PROGRAM P21_AL_WN
VAR
	//Analog Deviation Check
	Dev00, Dev01, Dev02, Dev03, Dev04, Dev05, Dev06, Dev07, Dev08, Dev09: FB_DeviationCheck;
	Dev10, Dev11, Dev12, Dev13, Dev14, Dev15, Dev16, Dev17, Dev18, Dev19: FB_DeviationCheck;
	Dev20, Dev21, Dev22, Dev23, Dev24, Dev25, Dev26, Dev27, Dev28, Dev29: FB_DeviationCheck;
		
	//Digital Noise Check
	wNoiseCheckTime: WORD := 100;	
	FB_AL32, FB_AL33, FB_AL34, FB_AL35, FB_AL36, FB_AL37, FB_AL38, FB_AL39: FB_NoiseCheck;	 
	FB_AL40, FB_AL41, FB_AL42, FB_AL43, FB_AL44, FB_AL45, FB_AL46, FB_AL47: FB_NoiseCheck;
	FB_AL48, FB_AL49, FB_AL50, FB_AL51, FB_AL52, FB_AL53, FB_AL54, FB_AL55: FB_NoiseCheck; 
	FB_AL56, FB_AL57, FB_AL58, FB_AL59, FB_AL60, FB_AL61, FB_AL62, FB_AL63: FB_NoiseCheck; 
	FB_AL64, FB_AL65, FB_AL66, FB_AL67, FB_AL68, FB_AL69, FB_AL70, FB_AL71: FB_NoiseCheck; 
	FB_AL72, FB_AL73, FB_AL74, FB_AL75, FB_AL76, FB_AL77, FB_AL78, FB_AL79: FB_NoiseCheck; 
	FB_AL80, FB_AL81, FB_AL82, FB_AL83, FB_AL84, FB_AL85, FB_AL86, FB_AL87: FB_NoiseCheck;
	FB_AL88, FB_AL89, FB_AL90, FB_AL91, FB_AL92, FB_AL93, FB_AL94, FB_AL95: FB_NoiseCheck; 
	FB_AL96, FB_AL97, FB_AL98, FB_AL99, FB_AL100, FB_AL101, FB_AL102, FB_AL103: FB_NoiseCheck; 
	FB_AL104, FB_AL105, FB_AL106, FB_AL107, FB_AL108, FB_AL109, FB_AL110, FB_AL111: FB_NoiseCheck;
	//FB_AL112, FB_AL113, FB_AL114, FB_AL115, FB_AL116, FB_AL117, FB_AL118, FB_AL119: FB_NoiseCheck; 
	FB_AL120, FB_AL121, FB_AL122, FB_AL123, FB_AL124, FB_AL125, FB_AL126, FB_AL127: FB_NoiseCheck;
	FB_AL128, FB_AL129, FB_AL130, FB_AL131, FB_AL132, FB_AL133, FB_AL134, FB_AL135: FB_NoiseCheck;
	FB_AL136, FB_AL137, FB_AL138, FB_AL139, FB_AL140, FB_AL141, FB_AL142, FB_AL143: FB_NoiseCheck;
	//FB_AL144, FB_AL145, FB_AL146, FB_AL147, FB_AL148, FB_AL149, FB_AL150, FB_AL151: FB_NoiseCheck;
	//FB_AL152, FB_AL153, FB_AL154, FB_AL155, FB_AL156, FB_AL157, FB_AL158, FB_AL159: FB_NoiseCheck;	
			
	FB_WN32, FB_WN33, FB_WN34, FB_WN35, FB_WN36, FB_WN37, FB_WN38, FB_WN39: FB_NoiseCheck; 
	FB_WN40, FB_WN41, FB_WN42, FB_WN43, FB_WN44, FB_WN45, FB_WN46, FB_WN47, FB_WN48, FB_WN49: FB_NoiseCheck; 
	FB_WN50, FB_WN51, FB_WN52, FB_WN53, FB_WN54, FB_WN55, FB_WN56, FB_WN57, FB_WN58, FB_WN59: FB_NoiseCheck; 
	FB_WN60, FB_WN61, FB_WN62, FB_WN63: FB_NoiseCheck;
									
	i: INT;
	bReset: BOOL;
	P_AL_Trig: R_TRIG;
	P_WN_Trig: R_TRIG;
	
	P_di_RST: R_TRIG;
		
	//Real Address
	n_AL_WORD AT%MB38: ARRAY[0..8] OF WORD; //16Bit
	n_WN_DWORD AT%MB56: ARRAY[0..1] OF DWORD; //32Bit
		
	n_AL_WORD_OLD: ARRAY[0..8] OF DWORD; //128EA
	n_WN_DWORD_OLD: ARRAY[0..1] OF DWORD; //64EA
	
	T1S_WN: TON;
	n_BZ_Order: ARRAY[0..1] OF BYTE;//부저 울림 순서, 1 -> Warning, 2 -> Alarm, 1 + 2 = 3 -> Alarm

END_VAR

A_AL_WN_Check();
D_AL_Check();
D_WN_Check();

is_AL := n_AL_WORD[0] > 0 OR n_AL_WORD[1] > 0 OR n_AL_WORD[2] > 0 OR n_AL_WORD[3] > 0 OR n_AL_WORD[4] > 0 OR
		 n_AL_WORD[5] > 0 OR n_AL_WORD[6] > 0 OR n_AL_WORD[7] > 0 OR n_AL_WORD[8] > 0;

is_WN := n_WN_DWORD[0] > 0 OR n_WN_DWORD[1] > 0 ;

//Alarm Processing
D_AL_Check();

//Alarm & Warning Reset
bReset := s_cm_RST;
 IF bReset THEN
	 s_is_DOR_Broken := 0;
 END_IF

//New AL Check
P_AL_Trig(CLK:= n_AL_WORD[0] > n_AL_WORD_OLD[0] OR n_AL_WORD[1] > n_AL_WORD_OLD[1] OR 
			  n_AL_WORD[2] > n_AL_WORD_OLD[2] OR n_AL_WORD[3] > n_AL_WORD_OLD[3] OR
			  n_AL_WORD[4] > n_AL_WORD_OLD[4] OR n_AL_WORD[5] > n_AL_WORD_OLD[5] OR
			  n_AL_WORD[6] > n_AL_WORD_OLD[6] OR n_AL_WORD[7] > n_AL_WORD_OLD[7] OR
			  n_AL_WORD[8] > n_AL_WORD_OLD[8]);
//New WN Check	
P_WN_Trig(CLK:= n_WN_DWORD[0] > n_WN_DWORD_OLD[0] OR n_WN_DWORD[1] > n_WN_DWORD_OLD[1]);

P_di_RST(CLK:= di_RST);	

//AL Backup	
FOR i := 0 TO 8 DO
	n_AL_WORD_OLD[i] := n_AL_WORD[i];
END_FOR
//WN Backup
FOR i := 0 TO 1 DO
	n_WN_DWORD_OLD[i] := n_WN_DWORD[i];
END_FOR

ACTION A_AL_WN_Check:
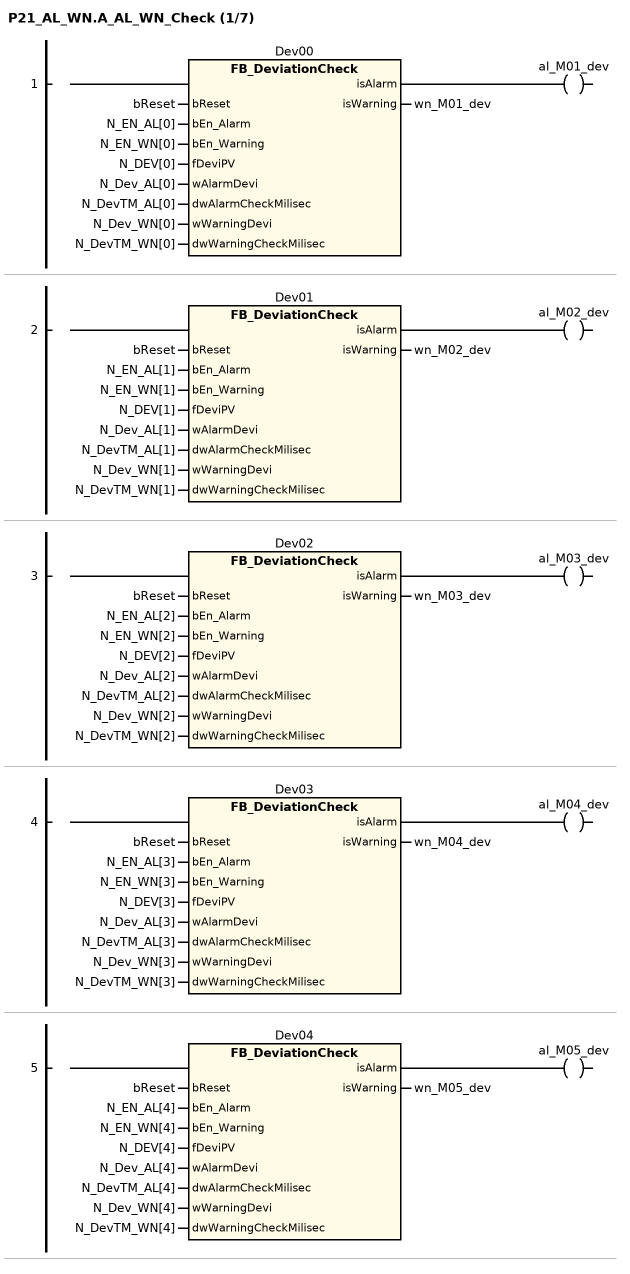
// NETWORK 1
Dev00(
    bReset := bReset,
    bEn_Alarm := N_EN_AL[0],
    bEn_Warning := N_EN_WN[0],
    fDeviPV := N_DEV[0],
    wAlarmDevi := N_Dev_AL[0],
    dwAlarmCheckMilisec := N_DevTM_AL[0],
    wWarningDevi := N_Dev_WN[0],
    dwWarningCheckMilisec := N_DevTM_WN[0],
    isWarning => wn_M01_dev); // FB_DeviationCheck
al_M01_dev := Dev00.isAlarm;

// NETWORK 2
Dev01(
    bReset := bReset,
    bEn_Alarm := N_EN_AL[1],
    bEn_Warning := N_EN_WN[1],
    fDeviPV := N_DEV[1],
    wAlarmDevi := N_Dev_AL[1],
    dwAlarmCheckMilisec := N_DevTM_AL[1],
    wWarningDevi := N_Dev_WN[1],
    dwWarningCheckMilisec := N_DevTM_WN[1],
    isWarning => wn_M02_dev); // FB_DeviationCheck
al_M02_dev := Dev01.isAlarm;

// NETWORK 3
Dev02(
    bReset := bReset,
    bEn_Alarm := N_EN_AL[2],
    bEn_Warning := N_EN_WN[2],
    fDeviPV := N_DEV[2],
    wAlarmDevi := N_Dev_AL[2],
    dwAlarmCheckMilisec := N_DevTM_AL[2],
    wWarningDevi := N_Dev_WN[2],
    dwWarningCheckMilisec := N_DevTM_WN[2],
    isWarning => wn_M03_dev); // FB_DeviationCheck
al_M03_dev := Dev02.isAlarm;

// NETWORK 4
Dev03(
    bReset := bReset,
    bEn_Alarm := N_EN_AL[3],
    bEn_Warning := N_EN_WN[3],
    fDeviPV := N_DEV[3],
    wAlarmDevi := N_Dev_AL[3],
    dwAlarmCheckMilisec := N_DevTM_AL[3],
    wWarningDevi := N_Dev_WN[3],
    dwWarningCheckMilisec := N_DevTM_WN[3],
    isWarning => wn_M04_dev); // FB_DeviationCheck
al_M04_dev := Dev03.isAlarm;

// NETWORK 5
Dev04(
    bReset := bReset,
    bEn_Alarm := N_EN_AL[4],
    bEn_Warning := N_EN_WN[4],
    fDeviPV := N_DEV[4],
    wAlarmDevi := N_Dev_AL[4],
    dwAlarmCheckMilisec := N_DevTM_AL[4],
    wWarningDevi := N_Dev_WN[4],
    dwWarningCheckMilisec := N_DevTM_WN[4],
    isWarning => wn_M05_dev); // FB_DeviationCheck
al_M05_dev := Dev04.isAlarm;

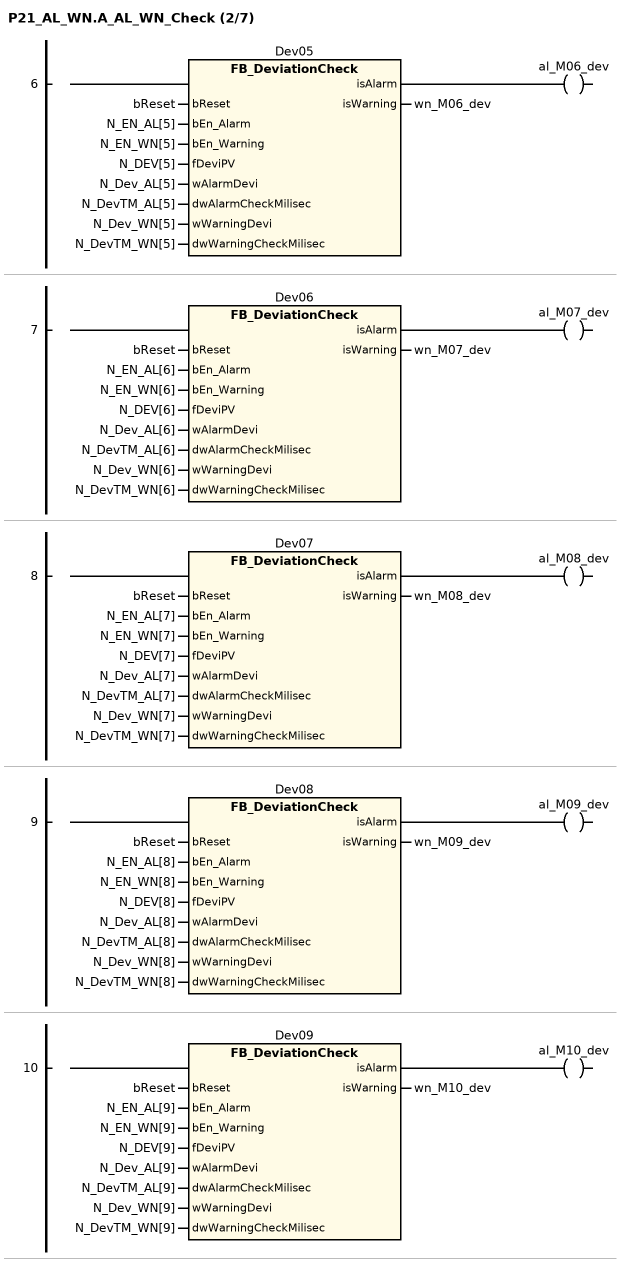
// NETWORK 6
Dev05(
    bReset := bReset,
    bEn_Alarm := N_EN_AL[5],
    bEn_Warning := N_EN_WN[5],
    fDeviPV := N_DEV[5],
    wAlarmDevi := N_Dev_AL[5],
    dwAlarmCheckMilisec := N_DevTM_AL[5],
    wWarningDevi := N_Dev_WN[5],
    dwWarningCheckMilisec := N_DevTM_WN[5],
    isWarning => wn_M06_dev); // FB_DeviationCheck
al_M06_dev := Dev05.isAlarm;

// NETWORK 7
Dev06(
    bReset := bReset,
    bEn_Alarm := N_EN_AL[6],
    bEn_Warning := N_EN_WN[6],
    fDeviPV := N_DEV[6],
    wAlarmDevi := N_Dev_AL[6],
    dwAlarmCheckMilisec := N_DevTM_AL[6],
    wWarningDevi := N_Dev_WN[6],
    dwWarningCheckMilisec := N_DevTM_WN[6],
    isWarning => wn_M07_dev); // FB_DeviationCheck
al_M07_dev := Dev06.isAlarm;

// NETWORK 8
Dev07(
    bReset := bReset,
    bEn_Alarm := N_EN_AL[7],
    bEn_Warning := N_EN_WN[7],
    fDeviPV := N_DEV[7],
    wAlarmDevi := N_Dev_AL[7],
    dwAlarmCheckMilisec := N_DevTM_AL[7],
    wWarningDevi := N_Dev_WN[7],
    dwWarningCheckMilisec := N_DevTM_WN[7],
    isWarning => wn_M08_dev); // FB_DeviationCheck
al_M08_dev := Dev07.isAlarm;

// NETWORK 9
Dev08(
    bReset := bReset,
    bEn_Alarm := N_EN_AL[8],
    bEn_Warning := N_EN_WN[8],
    fDeviPV := N_DEV[8],
    wAlarmDevi := N_Dev_AL[8],
    dwAlarmCheckMilisec := N_DevTM_AL[8],
    wWarningDevi := N_Dev_WN[8],
    dwWarningCheckMilisec := N_DevTM_WN[8],
    isWarning => wn_M09_dev); // FB_DeviationCheck
al_M09_dev := Dev08.isAlarm;

// NETWORK 10
Dev09(
    bReset := bReset,
    bEn_Alarm := N_EN_AL[9],
    bEn_Warning := N_EN_WN[9],
    fDeviPV := N_DEV[9],
    wAlarmDevi := N_Dev_AL[9],
    dwAlarmCheckMilisec := N_DevTM_AL[9],
    wWarningDevi := N_Dev_WN[9],
    dwWarningCheckMilisec := N_DevTM_WN[9],
    isWarning => wn_M10_dev); // FB_DeviationCheck
al_M10_dev := Dev09.isAlarm;

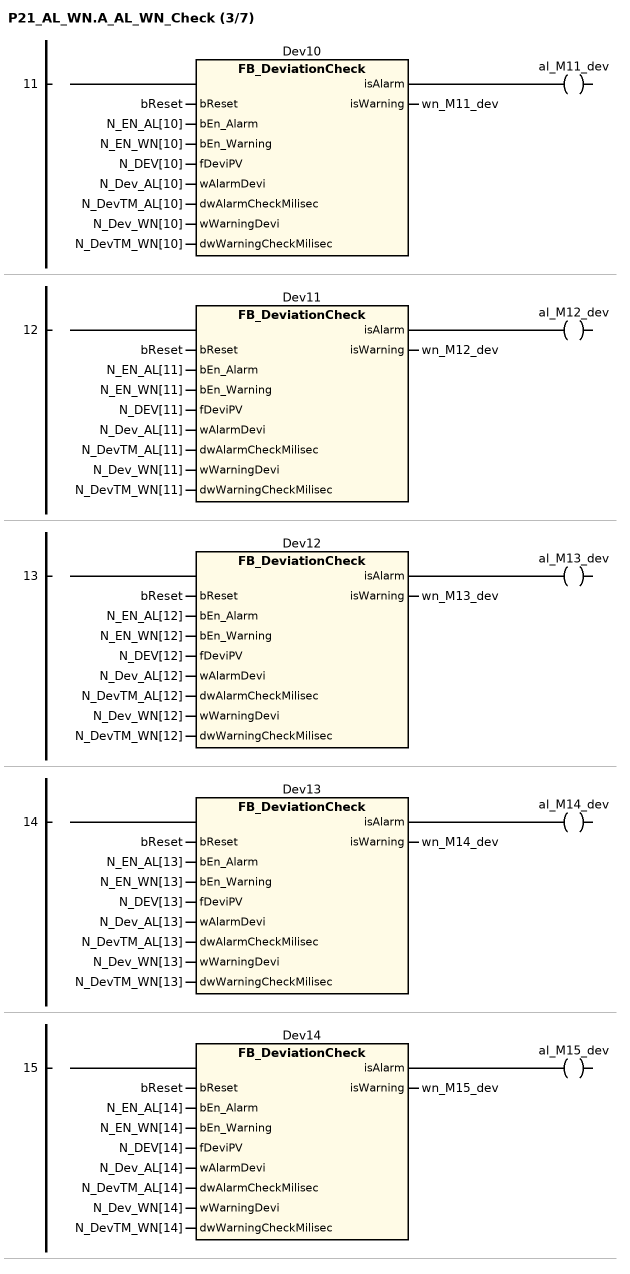
// NETWORK 11
Dev10(
    bReset := bReset,
    bEn_Alarm := N_EN_AL[10],
    bEn_Warning := N_EN_WN[10],
    fDeviPV := N_DEV[10],
    wAlarmDevi := N_Dev_AL[10],
    dwAlarmCheckMilisec := N_DevTM_AL[10],
    wWarningDevi := N_Dev_WN[10],
    dwWarningCheckMilisec := N_DevTM_WN[10],
    isWarning => wn_M11_dev); // FB_DeviationCheck
al_M11_dev := Dev10.isAlarm;

// NETWORK 12
Dev11(
    bReset := bReset,
    bEn_Alarm := N_EN_AL[11],
    bEn_Warning := N_EN_WN[11],
    fDeviPV := N_DEV[11],
    wAlarmDevi := N_Dev_AL[11],
    dwAlarmCheckMilisec := N_DevTM_AL[11],
    wWarningDevi := N_Dev_WN[11],
    dwWarningCheckMilisec := N_DevTM_WN[11],
    isWarning => wn_M12_dev); // FB_DeviationCheck
al_M12_dev := Dev11.isAlarm;

// NETWORK 13
Dev12(
    bReset := bReset,
    bEn_Alarm := N_EN_AL[12],
    bEn_Warning := N_EN_WN[12],
    fDeviPV := N_DEV[12],
    wAlarmDevi := N_Dev_AL[12],
    dwAlarmCheckMilisec := N_DevTM_AL[12],
    wWarningDevi := N_Dev_WN[12],
    dwWarningCheckMilisec := N_DevTM_WN[12],
    isWarning => wn_M13_dev); // FB_DeviationCheck
al_M13_dev := Dev12.isAlarm;

// NETWORK 14
Dev13(
    bReset := bReset,
    bEn_Alarm := N_EN_AL[13],
    bEn_Warning := N_EN_WN[13],
    fDeviPV := N_DEV[13],
    wAlarmDevi := N_Dev_AL[13],
    dwAlarmCheckMilisec := N_DevTM_AL[13],
    wWarningDevi := N_Dev_WN[13],
    dwWarningCheckMilisec := N_DevTM_WN[13],
    isWarning => wn_M14_dev); // FB_DeviationCheck
al_M14_dev := Dev13.isAlarm;

// NETWORK 15
Dev14(
    bReset := bReset,
    bEn_Alarm := N_EN_AL[14],
    bEn_Warning := N_EN_WN[14],
    fDeviPV := N_DEV[14],
    wAlarmDevi := N_Dev_AL[14],
    dwAlarmCheckMilisec := N_DevTM_AL[14],
    wWarningDevi := N_Dev_WN[14],
    dwWarningCheckMilisec := N_DevTM_WN[14],
    isWarning => wn_M15_dev); // FB_DeviationCheck
al_M15_dev := Dev14.isAlarm;

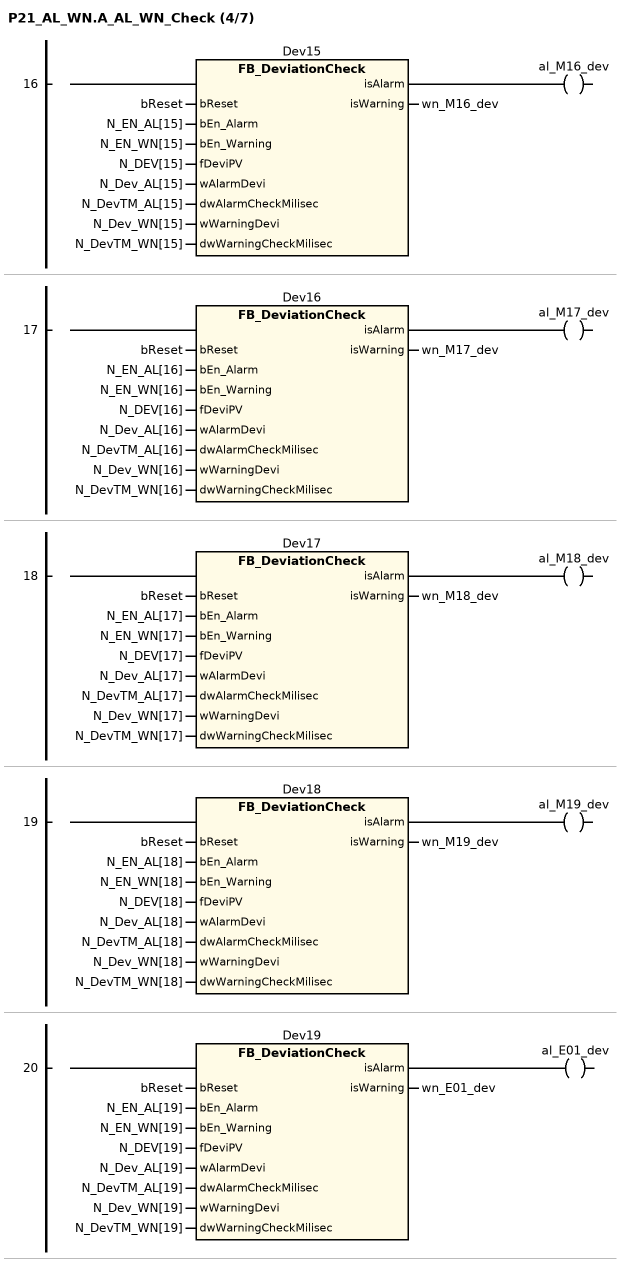
// NETWORK 16
Dev15(
    bReset := bReset,
    bEn_Alarm := N_EN_AL[15],
    bEn_Warning := N_EN_WN[15],
    fDeviPV := N_DEV[15],
    wAlarmDevi := N_Dev_AL[15],
    dwAlarmCheckMilisec := N_DevTM_AL[15],
    wWarningDevi := N_Dev_WN[15],
    dwWarningCheckMilisec := N_DevTM_WN[15],
    isWarning => wn_M16_dev); // FB_DeviationCheck
al_M16_dev := Dev15.isAlarm;

// NETWORK 17
Dev16(
    bReset := bReset,
    bEn_Alarm := N_EN_AL[16],
    bEn_Warning := N_EN_WN[16],
    fDeviPV := N_DEV[16],
    wAlarmDevi := N_Dev_AL[16],
    dwAlarmCheckMilisec := N_DevTM_AL[16],
    wWarningDevi := N_Dev_WN[16],
    dwWarningCheckMilisec := N_DevTM_WN[16],
    isWarning => wn_M17_dev); // FB_DeviationCheck
al_M17_dev := Dev16.isAlarm;

// NETWORK 18
Dev17(
    bReset := bReset,
    bEn_Alarm := N_EN_AL[17],
    bEn_Warning := N_EN_WN[17],
    fDeviPV := N_DEV[17],
    wAlarmDevi := N_Dev_AL[17],
    dwAlarmCheckMilisec := N_DevTM_AL[17],
    wWarningDevi := N_Dev_WN[17],
    dwWarningCheckMilisec := N_DevTM_WN[17],
    isWarning => wn_M18_dev); // FB_DeviationCheck
al_M18_dev := Dev17.isAlarm;

// NETWORK 19
Dev18(
    bReset := bReset,
    bEn_Alarm := N_EN_AL[18],
    bEn_Warning := N_EN_WN[18],
    fDeviPV := N_DEV[18],
    wAlarmDevi := N_Dev_AL[18],
    dwAlarmCheckMilisec := N_DevTM_AL[18],
    wWarningDevi := N_Dev_WN[18],
    dwWarningCheckMilisec := N_DevTM_WN[18],
    isWarning => wn_M19_dev); // FB_DeviationCheck
al_M19_dev := Dev18.isAlarm;

// NETWORK 20
Dev19(
    bReset := bReset,
    bEn_Alarm := N_EN_AL[19],
    bEn_Warning := N_EN_WN[19],
    fDeviPV := N_DEV[19],
    wAlarmDevi := N_Dev_AL[19],
    dwAlarmCheckMilisec := N_DevTM_AL[19],
    wWarningDevi := N_Dev_WN[19],
    dwWarningCheckMilisec := N_DevTM_WN[19],
    isWarning => wn_E01_dev); // FB_DeviationCheck
al_E01_dev := Dev19.isAlarm;

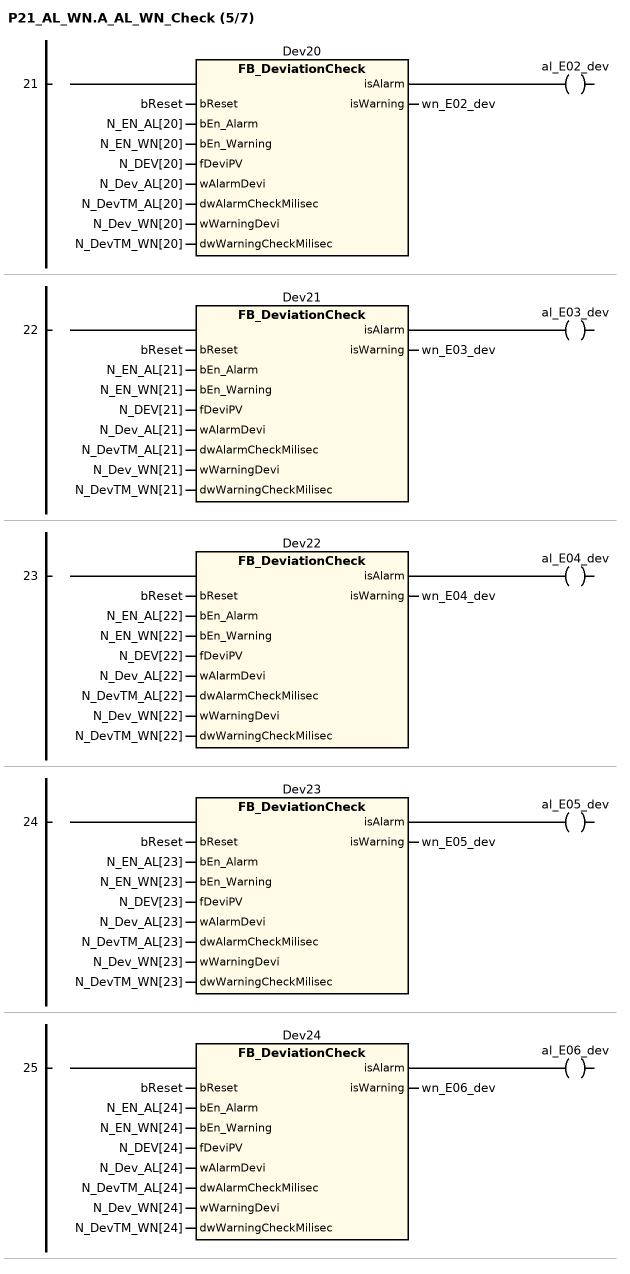
// NETWORK 21
Dev20(
    bReset := bReset,
    bEn_Alarm := N_EN_AL[20],
    bEn_Warning := N_EN_WN[20],
    fDeviPV := N_DEV[20],
    wAlarmDevi := N_Dev_AL[20],
    dwAlarmCheckMilisec := N_DevTM_AL[20],
    wWarningDevi := N_Dev_WN[20],
    dwWarningCheckMilisec := N_DevTM_WN[20],
    isWarning => wn_E02_dev); // FB_DeviationCheck
al_E02_dev := Dev20.isAlarm;

// NETWORK 22
Dev21(
    bReset := bReset,
    bEn_Alarm := N_EN_AL[21],
    bEn_Warning := N_EN_WN[21],
    fDeviPV := N_DEV[21],
    wAlarmDevi := N_Dev_AL[21],
    dwAlarmCheckMilisec := N_DevTM_AL[21],
    wWarningDevi := N_Dev_WN[21],
    dwWarningCheckMilisec := N_DevTM_WN[21],
    isWarning => wn_E03_dev); // FB_DeviationCheck
al_E03_dev := Dev21.isAlarm;

// NETWORK 23
Dev22(
    bReset := bReset,
    bEn_Alarm := N_EN_AL[22],
    bEn_Warning := N_EN_WN[22],
    fDeviPV := N_DEV[22],
    wAlarmDevi := N_Dev_AL[22],
    dwAlarmCheckMilisec := N_DevTM_AL[22],
    wWarningDevi := N_Dev_WN[22],
    dwWarningCheckMilisec := N_DevTM_WN[22],
    isWarning => wn_E04_dev); // FB_DeviationCheck
al_E04_dev := Dev22.isAlarm;

// NETWORK 24
Dev23(
    bReset := bReset,
    bEn_Alarm := N_EN_AL[23],
    bEn_Warning := N_EN_WN[23],
    fDeviPV := N_DEV[23],
    wAlarmDevi := N_Dev_AL[23],
    dwAlarmCheckMilisec := N_DevTM_AL[23],
    wWarningDevi := N_Dev_WN[23],
    dwWarningCheckMilisec := N_DevTM_WN[23],
    isWarning => wn_E05_dev); // FB_DeviationCheck
al_E05_dev := Dev23.isAlarm;

// NETWORK 25
Dev24(
    bReset := bReset,
    bEn_Alarm := N_EN_AL[24],
    bEn_Warning := N_EN_WN[24],
    fDeviPV := N_DEV[24],
    wAlarmDevi := N_Dev_AL[24],
    dwAlarmCheckMilisec := N_DevTM_AL[24],
    wWarningDevi := N_Dev_WN[24],
    dwWarningCheckMilisec := N_DevTM_WN[24],
    isWarning => wn_E06_dev); // FB_DeviationCheck
al_E06_dev := Dev24.isAlarm;

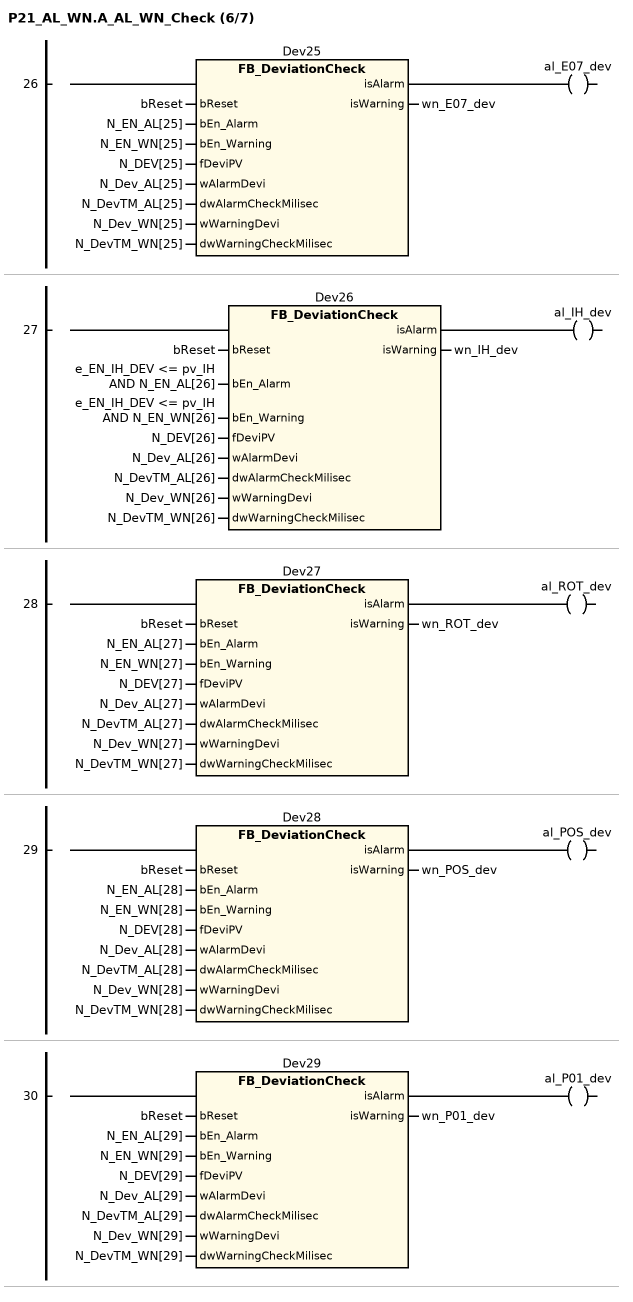
// NETWORK 26
Dev25(
    bReset := bReset,
    bEn_Alarm := N_EN_AL[25],
    bEn_Warning := N_EN_WN[25],
    fDeviPV := N_DEV[25],
    wAlarmDevi := N_Dev_AL[25],
    dwAlarmCheckMilisec := N_DevTM_AL[25],
    wWarningDevi := N_Dev_WN[25],
    dwWarningCheckMilisec := N_DevTM_WN[25],
    isWarning => wn_E07_dev); // FB_DeviationCheck
al_E07_dev := Dev25.isAlarm;

// NETWORK 27
Dev26(
    bReset := bReset,
    bEn_Alarm := e_EN_IH_DEV <= pv_IH AND N_EN_AL[26],
    bEn_Warning := e_EN_IH_DEV <= pv_IH AND N_EN_WN[26],
    fDeviPV := N_DEV[26],
    wAlarmDevi := N_Dev_AL[26],
    dwAlarmCheckMilisec := N_DevTM_AL[26],
    wWarningDevi := N_Dev_WN[26],
    dwWarningCheckMilisec := N_DevTM_WN[26],
    isWarning => wn_IH_dev); // FB_DeviationCheck
al_IH_dev := Dev26.isAlarm;

// NETWORK 28
Dev27(
    bReset := bReset,
    bEn_Alarm := N_EN_AL[27],
    bEn_Warning := N_EN_WN[27],
    fDeviPV := N_DEV[27],
    wAlarmDevi := N_Dev_AL[27],
    dwAlarmCheckMilisec := N_DevTM_AL[27],
    wWarningDevi := N_Dev_WN[27],
    dwWarningCheckMilisec := N_DevTM_WN[27],
    isWarning => wn_ROT_dev); // FB_DeviationCheck
al_ROT_dev := Dev27.isAlarm;

// NETWORK 29
Dev28(
    bReset := bReset,
    bEn_Alarm := N_EN_AL[28],
    bEn_Warning := N_EN_WN[28],
    fDeviPV := N_DEV[28],
    wAlarmDevi := N_Dev_AL[28],
    dwAlarmCheckMilisec := N_DevTM_AL[28],
    wWarningDevi := N_Dev_WN[28],
    dwWarningCheckMilisec := N_DevTM_WN[28],
    isWarning => wn_POS_dev); // FB_DeviationCheck
al_POS_dev := Dev28.isAlarm;

// NETWORK 30
Dev29(
    bReset := bReset,
    bEn_Alarm := N_EN_AL[29],
    bEn_Warning := N_EN_WN[29],
    fDeviPV := N_DEV[29],
    wAlarmDevi := N_Dev_AL[29],
    dwAlarmCheckMilisec := N_DevTM_AL[29],
    wWarningDevi := N_Dev_WN[29],
    dwWarningCheckMilisec := N_DevTM_WN[29],
    isWarning => wn_P01_dev); // FB_DeviationCheck
al_P01_dev := Dev29.isAlarm;

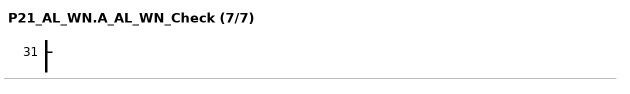
// NETWORK 31
END_ACTION

ACTION Cause_N_Effect:

//WN Buzzer
IF P_WN_Trig.Q THEN
	IF n_BZ_Order[0] <= 0 THEN
		n_BZ_Order[0] := 1; 
	ELSE
		IF n_BZ_Order[0] <> 1 THEN
			n_BZ_Order[1] := 1;
		END_IF
	END_IF
END_IF

//new Alarm rised
IF P_AL_Trig.Q THEN	
	//AL Buzzer
	IF n_BZ_Order[0] <= 0 THEN
		n_BZ_Order[0] := 2; 
	ELSE
		IF n_BZ_Order[0] <> 2 THEN
			n_BZ_Order[1] := 2;
		END_IF
	END_IF
	//AL UserState	
	IF e_US_AL > 0 THEN
		CASE e_US_AL OF
			1: cm_US1 := 1;
			2: cm_US2 := 1;
			3: cm_US3 := 1;
			4: cm_US4 := 1;
		END_CASE
	END_IF	
END_IF	

//IHT 
IF al_PCW_low OR al_IH_fail OR al_IH_overT OR al_SH_CW_overT OR al_IH_CW_overT THEN
	cm_IH := 0;
END_IF
					 
//H2 & SiH4 & NH3
IF is_AL THEN	
	cm_V01 := 0;// H2 Supply
	cm_V02 := 0;// H2 Supply
	cm_V03 := 0;//SiH4 Supply
	cm_V04 := 0;//NH3 Supply
END_IF

IF is_P01_overP_al THEN //둘다 닫아 자연스럽게 동자
	cm_V33_1 := 0;
	cm_V33_2 := 0;
END_IF

IF al_DOR OR wn_DOR THEN
	s_DOR_CNT := 0;
END_IF


//Buzzer Off Process
IF cm_BZ_UserStop OR P_di_RST.Q THEN
	IF n_BZ_Order[0] > 0 THEN
		n_BZ_Order[0] := 0; 
	ELSE
		n_BZ_Order[1] := 0;
	END_IF
	cm_BZ := 0;
	cm_BZ_UserStop := 0; 
END_IF

//Buzzer On Process
IF ing_Maint = 0 THEN	
	T1S_WN(PT:=T#1S);
	T1S_WN.IN :=  n_BZ_Order[0] + n_BZ_Order[1] = 1;
	IF T1S_WN.Q THEN //warning buzzer is 1sec cycle
		T1S_WN.IN := 0;
		cm_BZ := NOT cm_BZ;
	END_IF
	
	IF n_BZ_Order[0] + n_BZ_Order[1] >= 2 THEN
		cm_BZ := 1;
	END_IF
END_IF


//H2	
//IF al_N2_Low OR  al_H2_Low OR al_NH3_Low OR al_GC_H2_Leak OR al_RC_H2_Leak  THEN 
	//H2 Valve OFF - kjk??
	//cm_V27 := OFF;
//END_IF

//EMG_InductionPower
(*IF al_CW_IH_TempHi = ON THEN
	do_IH_Pow := OFF;
ELSE
	IF al_CHM_TempHi = ON THEN
		do_IH_Pow := OFF;
	ELSE
		IF al_GC_H2_Leak = ON THEN
			do_IH_Pow := OFF;
		ELSE
			IF al_RC_H2_Leak = ON THEN
				do_IH_Pow := OFF;
			ELSE
				do_IH_Pow := ON;	
			END_IF		
		END_IF		
	END_IF		
END_IF *)
END_ACTION

ACTION D_AL_Check:
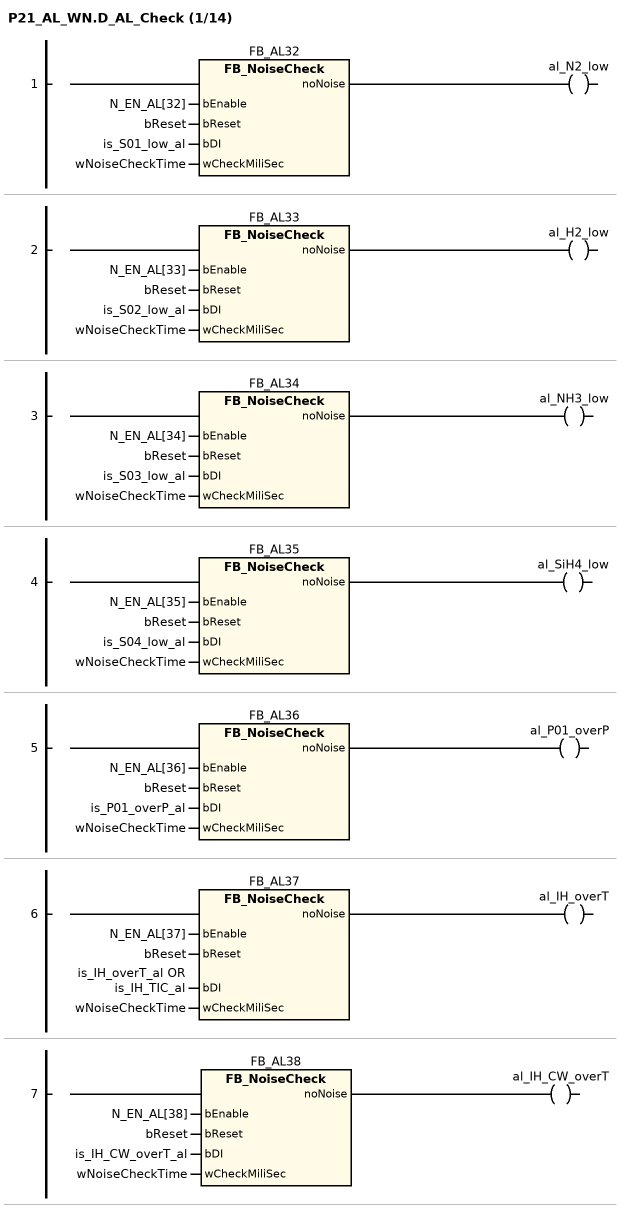
// NETWORK 1
FB_AL32(bEnable := N_EN_AL[32], bReset := bReset, bDI := is_S01_low_al, wCheckMiliSec := wNoiseCheckTime); // FB_NoiseCheck
al_N2_low := FB_AL32.noNoise;

// NETWORK 2
FB_AL33(bEnable := N_EN_AL[33], bReset := bReset, bDI := is_S02_low_al, wCheckMiliSec := wNoiseCheckTime); // FB_NoiseCheck
al_H2_low := FB_AL33.noNoise;

// NETWORK 3
FB_AL34(bEnable := N_EN_AL[34], bReset := bReset, bDI := is_S03_low_al, wCheckMiliSec := wNoiseCheckTime); // FB_NoiseCheck
al_NH3_low := FB_AL34.noNoise;

// NETWORK 4
FB_AL35(bEnable := N_EN_AL[35], bReset := bReset, bDI := is_S04_low_al, wCheckMiliSec := wNoiseCheckTime); // FB_NoiseCheck
al_SiH4_low := FB_AL35.noNoise;

// NETWORK 5
FB_AL36(bEnable := N_EN_AL[36], bReset := bReset, bDI := is_P01_overP_al, wCheckMiliSec := wNoiseCheckTime); // FB_NoiseCheck
al_P01_overP := FB_AL36.noNoise;

// NETWORK 6
FB_AL37(
    bEnable := N_EN_AL[37],
    bReset := bReset,
    bDI := is_IH_overT_al OR is_IH_TIC_al,
    wCheckMiliSec := wNoiseCheckTime); // FB_NoiseCheck
al_IH_overT := FB_AL37.noNoise;

// NETWORK 7
FB_AL38(bEnable := N_EN_AL[38], bReset := bReset, bDI := is_IH_CW_overT_al, wCheckMiliSec := wNoiseCheckTime); // FB_NoiseCheck
al_IH_CW_overT := FB_AL38.noNoise;

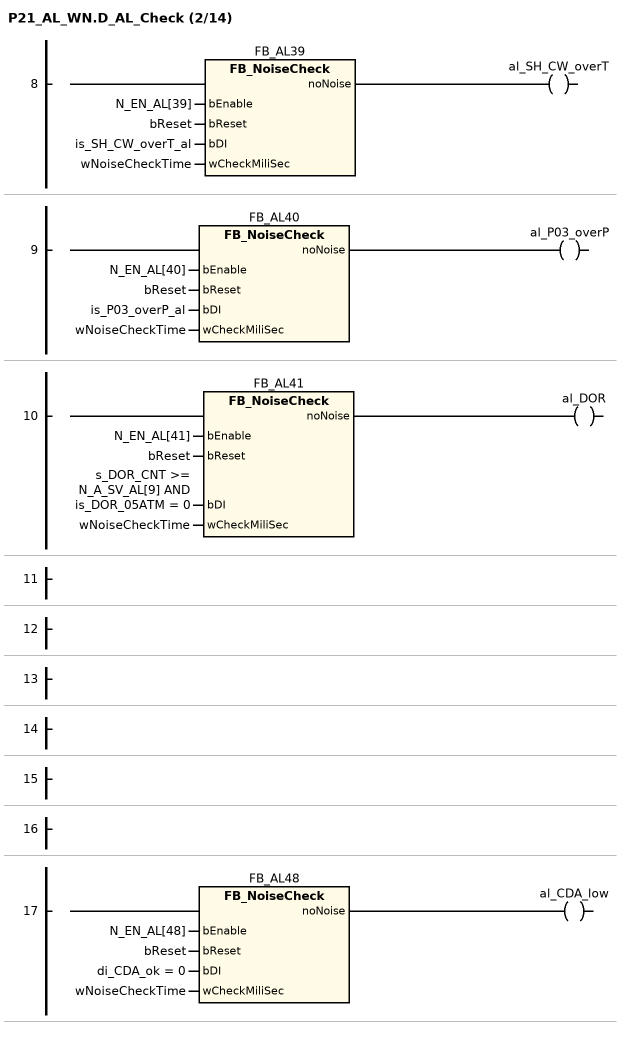
// NETWORK 8
FB_AL39(bEnable := N_EN_AL[39], bReset := bReset, bDI := is_SH_CW_overT_al, wCheckMiliSec := wNoiseCheckTime); // FB_NoiseCheck
al_SH_CW_overT := FB_AL39.noNoise;

// NETWORK 9
FB_AL40(bEnable := N_EN_AL[40], bReset := bReset, bDI := is_P03_overP_al, wCheckMiliSec := wNoiseCheckTime); // FB_NoiseCheck
al_P03_overP := FB_AL40.noNoise;

// NETWORK 10
FB_AL41(
    bEnable := N_EN_AL[41],
    bReset := bReset,
    bDI := s_DOR_CNT >= N_A_SV_AL[9] AND is_DOR_05ATM = 0,
    wCheckMiliSec := wNoiseCheckTime); // FB_NoiseCheck
al_DOR := FB_AL41.noNoise;

// NETWORK 11

// NETWORK 12

// NETWORK 13

// NETWORK 14

// NETWORK 15

// NETWORK 16

// NETWORK 17
FB_AL48(bEnable := N_EN_AL[48], bReset := bReset, bDI := di_CDA_ok = 0, wCheckMiliSec := wNoiseCheckTime); // FB_NoiseCheck
al_CDA_low := FB_AL48.noNoise;

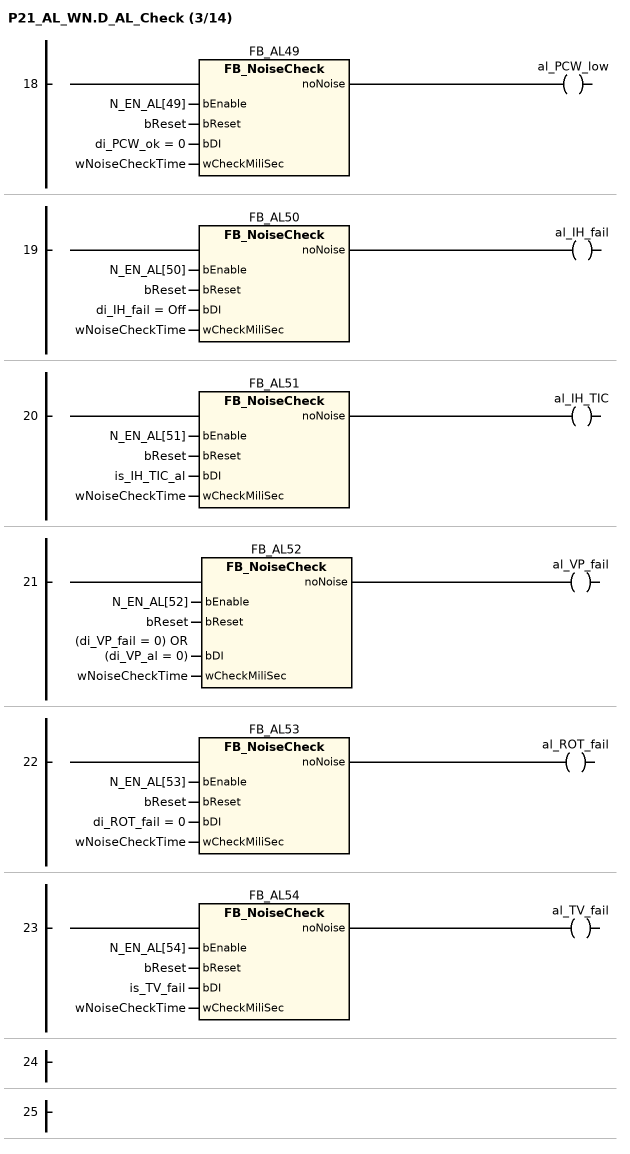
// NETWORK 18
FB_AL49(bEnable := N_EN_AL[49], bReset := bReset, bDI := di_PCW_ok = 0, wCheckMiliSec := wNoiseCheckTime); // FB_NoiseCheck
al_PCW_low := FB_AL49.noNoise;

// NETWORK 19
FB_AL50(bEnable := N_EN_AL[50], bReset := bReset, bDI := di_IH_fail = Off, wCheckMiliSec := wNoiseCheckTime); // FB_NoiseCheck
al_IH_fail := FB_AL50.noNoise;

// NETWORK 20
FB_AL51(bEnable := N_EN_AL[51], bReset := bReset, bDI := is_IH_TIC_al, wCheckMiliSec := wNoiseCheckTime); // FB_NoiseCheck
al_IH_TIC := FB_AL51.noNoise;

// NETWORK 21
FB_AL52(
    bEnable := N_EN_AL[52],
    bReset := bReset,
    bDI := (di_VP_fail = 0) OR (di_VP_al = 0),
    wCheckMiliSec := wNoiseCheckTime); // FB_NoiseCheck
al_VP_fail := FB_AL52.noNoise;

// NETWORK 22
FB_AL53(bEnable := N_EN_AL[53], bReset := bReset, bDI := di_ROT_fail = 0, wCheckMiliSec := wNoiseCheckTime); // FB_NoiseCheck
al_ROT_fail := FB_AL53.noNoise;

// NETWORK 23
FB_AL54(bEnable := N_EN_AL[54], bReset := bReset, bDI := is_TV_fail, wCheckMiliSec := wNoiseCheckTime); // FB_NoiseCheck
al_TV_fail := FB_AL54.noNoise;

// NETWORK 24

// NETWORK 25

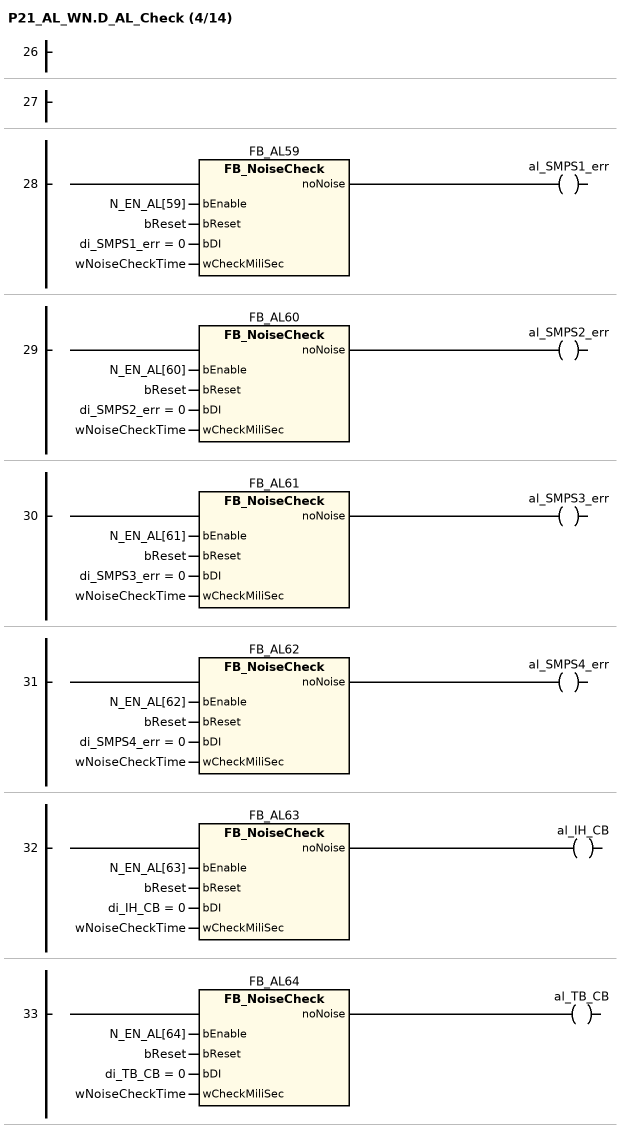
// NETWORK 26

// NETWORK 27

// NETWORK 28
FB_AL59(bEnable := N_EN_AL[59], bReset := bReset, bDI := di_SMPS1_err = 0, wCheckMiliSec := wNoiseCheckTime); // FB_NoiseCheck
al_SMPS1_err := FB_AL59.noNoise;

// NETWORK 29
FB_AL60(bEnable := N_EN_AL[60], bReset := bReset, bDI := di_SMPS2_err = 0, wCheckMiliSec := wNoiseCheckTime); // FB_NoiseCheck
al_SMPS2_err := FB_AL60.noNoise;

// NETWORK 30
FB_AL61(bEnable := N_EN_AL[61], bReset := bReset, bDI := di_SMPS3_err = 0, wCheckMiliSec := wNoiseCheckTime); // FB_NoiseCheck
al_SMPS3_err := FB_AL61.noNoise;

// NETWORK 31
FB_AL62(bEnable := N_EN_AL[62], bReset := bReset, bDI := di_SMPS4_err = 0, wCheckMiliSec := wNoiseCheckTime); // FB_NoiseCheck
al_SMPS4_err := FB_AL62.noNoise;

// NETWORK 32
FB_AL63(bEnable := N_EN_AL[63], bReset := bReset, bDI := di_IH_CB = 0, wCheckMiliSec := wNoiseCheckTime); // FB_NoiseCheck
al_IH_CB := FB_AL63.noNoise;

// NETWORK 33
FB_AL64(bEnable := N_EN_AL[64], bReset := bReset, bDI := di_TB_CB = 0, wCheckMiliSec := wNoiseCheckTime); // FB_NoiseCheck
al_TB_CB := FB_AL64.noNoise;

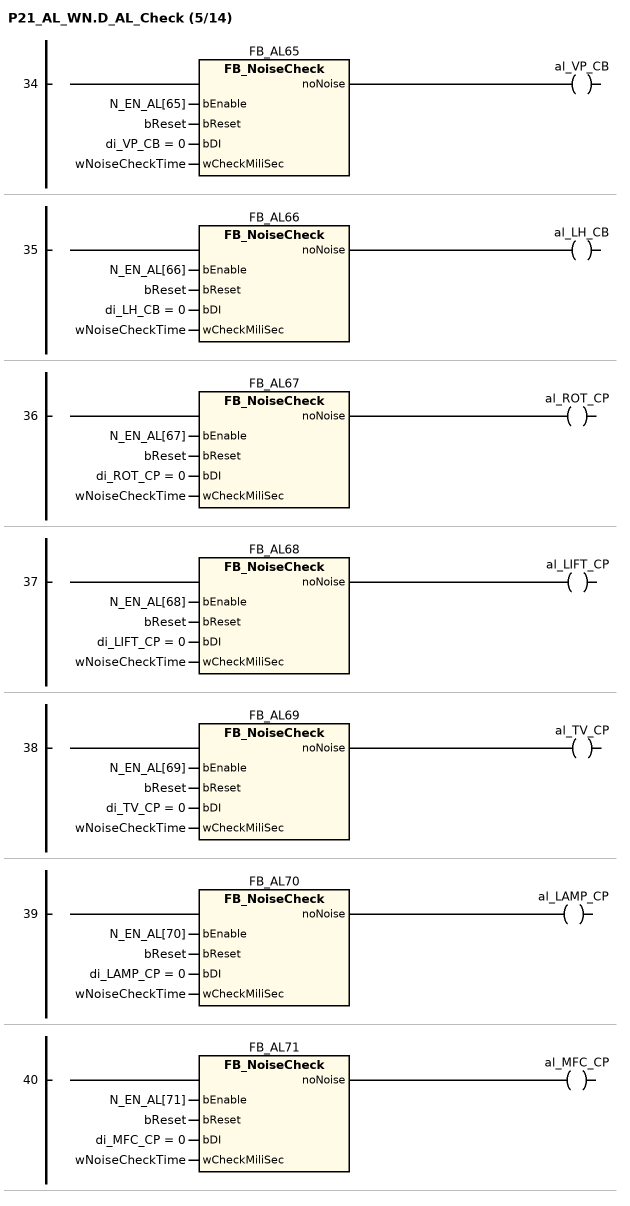
// NETWORK 34
FB_AL65(bEnable := N_EN_AL[65], bReset := bReset, bDI := di_VP_CB = 0, wCheckMiliSec := wNoiseCheckTime); // FB_NoiseCheck
al_VP_CB := FB_AL65.noNoise;

// NETWORK 35
FB_AL66(bEnable := N_EN_AL[66], bReset := bReset, bDI := di_LH_CB = 0, wCheckMiliSec := wNoiseCheckTime); // FB_NoiseCheck
al_LH_CB := FB_AL66.noNoise;

// NETWORK 36
FB_AL67(bEnable := N_EN_AL[67], bReset := bReset, bDI := di_ROT_CP = 0, wCheckMiliSec := wNoiseCheckTime); // FB_NoiseCheck
al_ROT_CP := FB_AL67.noNoise;

// NETWORK 37
FB_AL68(bEnable := N_EN_AL[68], bReset := bReset, bDI := di_LIFT_CP = 0, wCheckMiliSec := wNoiseCheckTime); // FB_NoiseCheck
al_LIFT_CP := FB_AL68.noNoise;

// NETWORK 38
FB_AL69(bEnable := N_EN_AL[69], bReset := bReset, bDI := di_TV_CP = 0, wCheckMiliSec := wNoiseCheckTime); // FB_NoiseCheck
al_TV_CP := FB_AL69.noNoise;

// NETWORK 39
FB_AL70(bEnable := N_EN_AL[70], bReset := bReset, bDI := di_LAMP_CP = 0, wCheckMiliSec := wNoiseCheckTime); // FB_NoiseCheck
al_LAMP_CP := FB_AL70.noNoise;

// NETWORK 40
FB_AL71(bEnable := N_EN_AL[71], bReset := bReset, bDI := di_MFC_CP = 0, wCheckMiliSec := wNoiseCheckTime); // FB_NoiseCheck
al_MFC_CP := FB_AL71.noNoise;

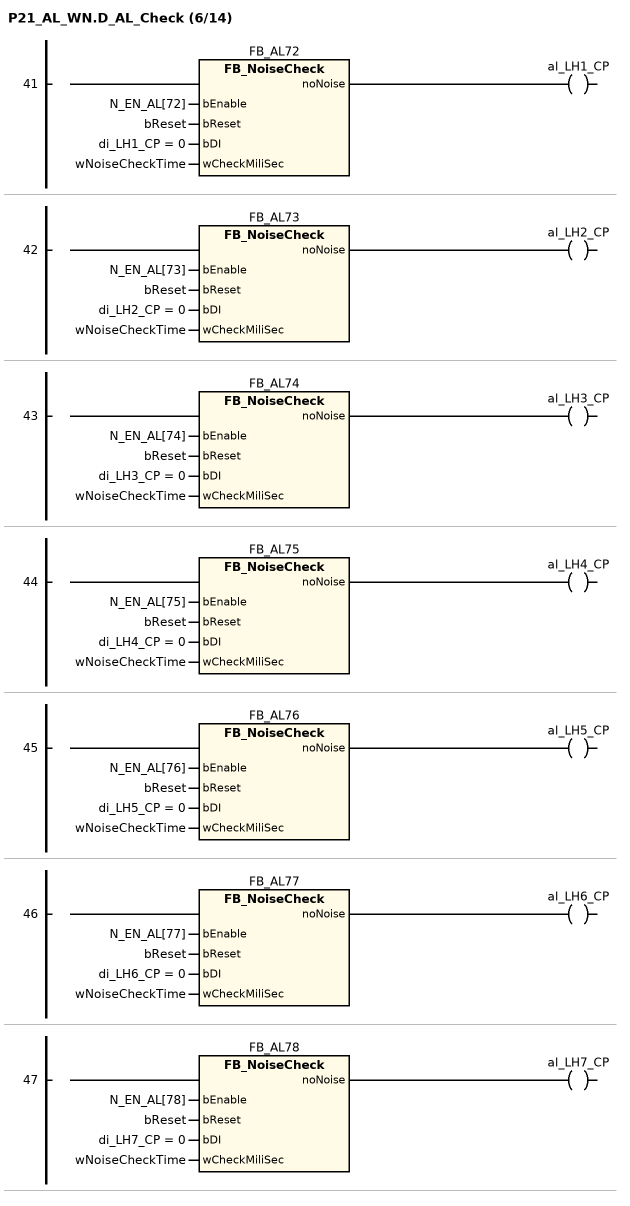
// NETWORK 41
FB_AL72(bEnable := N_EN_AL[72], bReset := bReset, bDI := di_LH1_CP = 0, wCheckMiliSec := wNoiseCheckTime); // FB_NoiseCheck
al_LH1_CP := FB_AL72.noNoise;

// NETWORK 42
FB_AL73(bEnable := N_EN_AL[73], bReset := bReset, bDI := di_LH2_CP = 0, wCheckMiliSec := wNoiseCheckTime); // FB_NoiseCheck
al_LH2_CP := FB_AL73.noNoise;

// NETWORK 43
FB_AL74(bEnable := N_EN_AL[74], bReset := bReset, bDI := di_LH3_CP = 0, wCheckMiliSec := wNoiseCheckTime); // FB_NoiseCheck
al_LH3_CP := FB_AL74.noNoise;

// NETWORK 44
FB_AL75(bEnable := N_EN_AL[75], bReset := bReset, bDI := di_LH4_CP = 0, wCheckMiliSec := wNoiseCheckTime); // FB_NoiseCheck
al_LH4_CP := FB_AL75.noNoise;

// NETWORK 45
FB_AL76(bEnable := N_EN_AL[76], bReset := bReset, bDI := di_LH5_CP = 0, wCheckMiliSec := wNoiseCheckTime); // FB_NoiseCheck
al_LH5_CP := FB_AL76.noNoise;

// NETWORK 46
FB_AL77(bEnable := N_EN_AL[77], bReset := bReset, bDI := di_LH6_CP = 0, wCheckMiliSec := wNoiseCheckTime); // FB_NoiseCheck
al_LH6_CP := FB_AL77.noNoise;

// NETWORK 47
FB_AL78(bEnable := N_EN_AL[78], bReset := bReset, bDI := di_LH7_CP = 0, wCheckMiliSec := wNoiseCheckTime); // FB_NoiseCheck
al_LH7_CP := FB_AL78.noNoise;

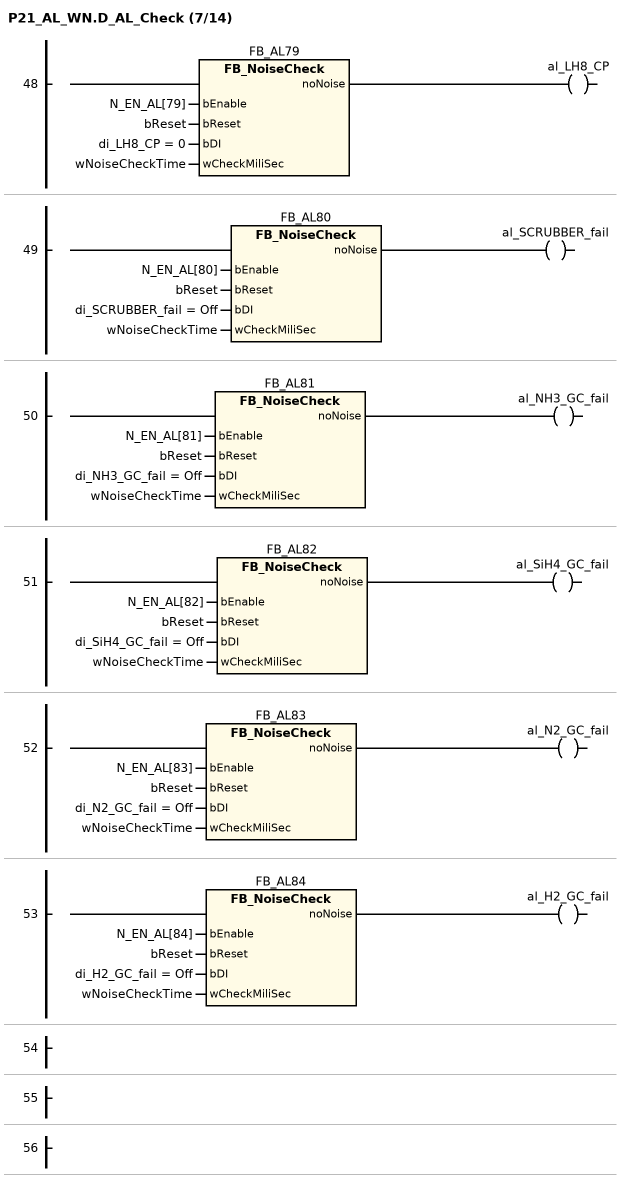
// NETWORK 48
FB_AL79(bEnable := N_EN_AL[79], bReset := bReset, bDI := di_LH8_CP = 0, wCheckMiliSec := wNoiseCheckTime); // FB_NoiseCheck
al_LH8_CP := FB_AL79.noNoise;

// NETWORK 49
FB_AL80(
    bEnable := N_EN_AL[80],
    bReset := bReset,
    bDI := di_SCRUBBER_fail = Off,
    wCheckMiliSec := wNoiseCheckTime); // FB_NoiseCheck
al_SCRUBBER_fail := FB_AL80.noNoise;

// NETWORK 50
FB_AL81(
    bEnable := N_EN_AL[81],
    bReset := bReset,
    bDI := di_NH3_GC_fail = Off,
    wCheckMiliSec := wNoiseCheckTime); // FB_NoiseCheck
al_NH3_GC_fail := FB_AL81.noNoise;

// NETWORK 51
FB_AL82(
    bEnable := N_EN_AL[82],
    bReset := bReset,
    bDI := di_SiH4_GC_fail = Off,
    wCheckMiliSec := wNoiseCheckTime); // FB_NoiseCheck
al_SiH4_GC_fail := FB_AL82.noNoise;

// NETWORK 52
FB_AL83(
    bEnable := N_EN_AL[83],
    bReset := bReset,
    bDI := di_N2_GC_fail = Off,
    wCheckMiliSec := wNoiseCheckTime); // FB_NoiseCheck
al_N2_GC_fail := FB_AL83.noNoise;

// NETWORK 53
FB_AL84(
    bEnable := N_EN_AL[84],
    bReset := bReset,
    bDI := di_H2_GC_fail = Off,
    wCheckMiliSec := wNoiseCheckTime); // FB_NoiseCheck
al_H2_GC_fail := FB_AL84.noNoise;

// NETWORK 54

// NETWORK 55

// NETWORK 56

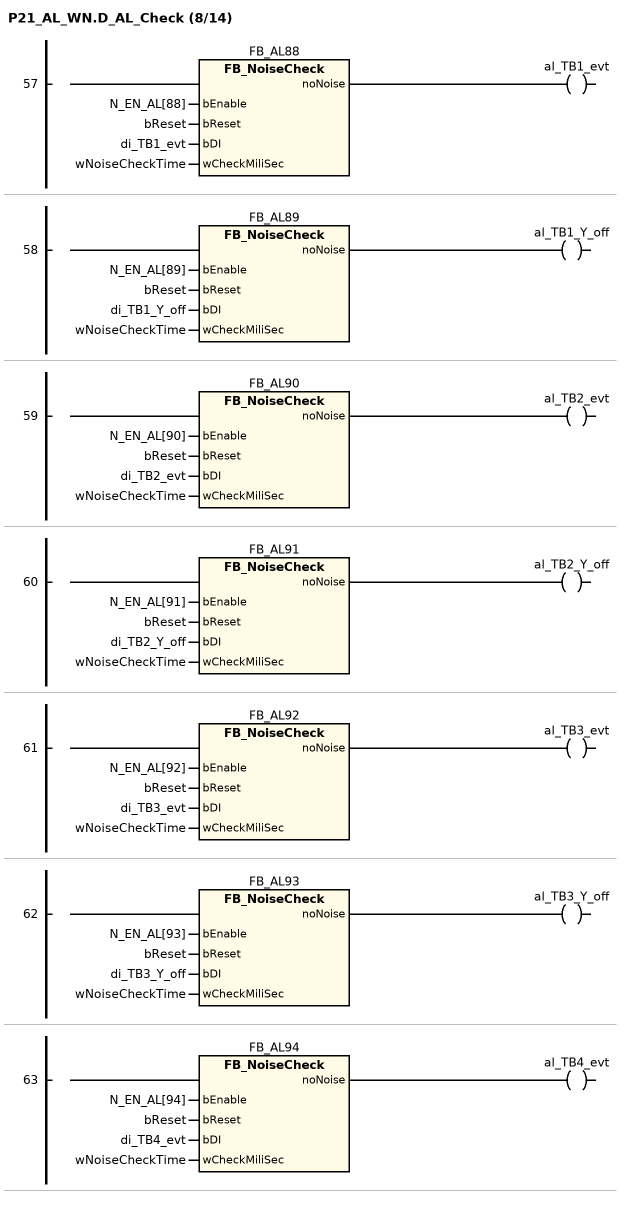
// NETWORK 57
FB_AL88(bEnable := N_EN_AL[88], bReset := bReset, bDI := di_TB1_evt, wCheckMiliSec := wNoiseCheckTime); // FB_NoiseCheck
al_TB1_evt := FB_AL88.noNoise;

// NETWORK 58
FB_AL89(bEnable := N_EN_AL[89], bReset := bReset, bDI := di_TB1_Y_off, wCheckMiliSec := wNoiseCheckTime); // FB_NoiseCheck
al_TB1_Y_off := FB_AL89.noNoise;

// NETWORK 59
FB_AL90(bEnable := N_EN_AL[90], bReset := bReset, bDI := di_TB2_evt, wCheckMiliSec := wNoiseCheckTime); // FB_NoiseCheck
al_TB2_evt := FB_AL90.noNoise;

// NETWORK 60
FB_AL91(bEnable := N_EN_AL[91], bReset := bReset, bDI := di_TB2_Y_off, wCheckMiliSec := wNoiseCheckTime); // FB_NoiseCheck
al_TB2_Y_off := FB_AL91.noNoise;

// NETWORK 61
FB_AL92(bEnable := N_EN_AL[92], bReset := bReset, bDI := di_TB3_evt, wCheckMiliSec := wNoiseCheckTime); // FB_NoiseCheck
al_TB3_evt := FB_AL92.noNoise;

// NETWORK 62
FB_AL93(bEnable := N_EN_AL[93], bReset := bReset, bDI := di_TB3_Y_off, wCheckMiliSec := wNoiseCheckTime); // FB_NoiseCheck
al_TB3_Y_off := FB_AL93.noNoise;

// NETWORK 63
FB_AL94(bEnable := N_EN_AL[94], bReset := bReset, bDI := di_TB4_evt, wCheckMiliSec := wNoiseCheckTime); // FB_NoiseCheck
al_TB4_evt := FB_AL94.noNoise;

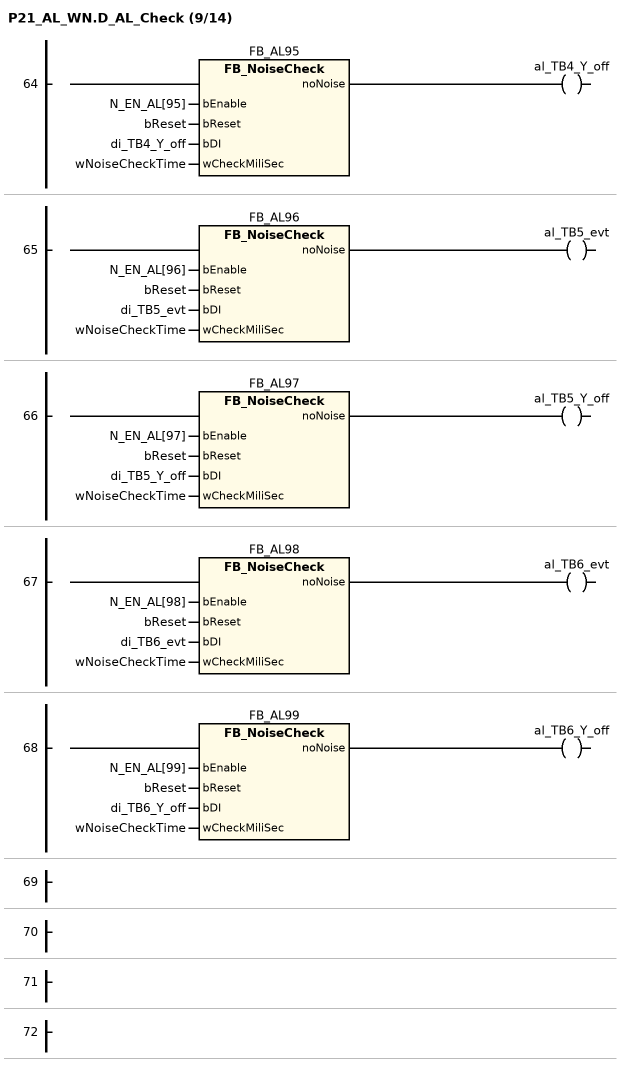
// NETWORK 64
FB_AL95(bEnable := N_EN_AL[95], bReset := bReset, bDI := di_TB4_Y_off, wCheckMiliSec := wNoiseCheckTime); // FB_NoiseCheck
al_TB4_Y_off := FB_AL95.noNoise;

// NETWORK 65
FB_AL96(bEnable := N_EN_AL[96], bReset := bReset, bDI := di_TB5_evt, wCheckMiliSec := wNoiseCheckTime); // FB_NoiseCheck
al_TB5_evt := FB_AL96.noNoise;

// NETWORK 66
FB_AL97(bEnable := N_EN_AL[97], bReset := bReset, bDI := di_TB5_Y_off, wCheckMiliSec := wNoiseCheckTime); // FB_NoiseCheck
al_TB5_Y_off := FB_AL97.noNoise;

// NETWORK 67
FB_AL98(bEnable := N_EN_AL[98], bReset := bReset, bDI := di_TB6_evt, wCheckMiliSec := wNoiseCheckTime); // FB_NoiseCheck
al_TB6_evt := FB_AL98.noNoise;

// NETWORK 68
FB_AL99(bEnable := N_EN_AL[99], bReset := bReset, bDI := di_TB6_Y_off, wCheckMiliSec := wNoiseCheckTime); // FB_NoiseCheck
al_TB6_Y_off := FB_AL99.noNoise;

// NETWORK 69

// NETWORK 70

// NETWORK 71

// NETWORK 72

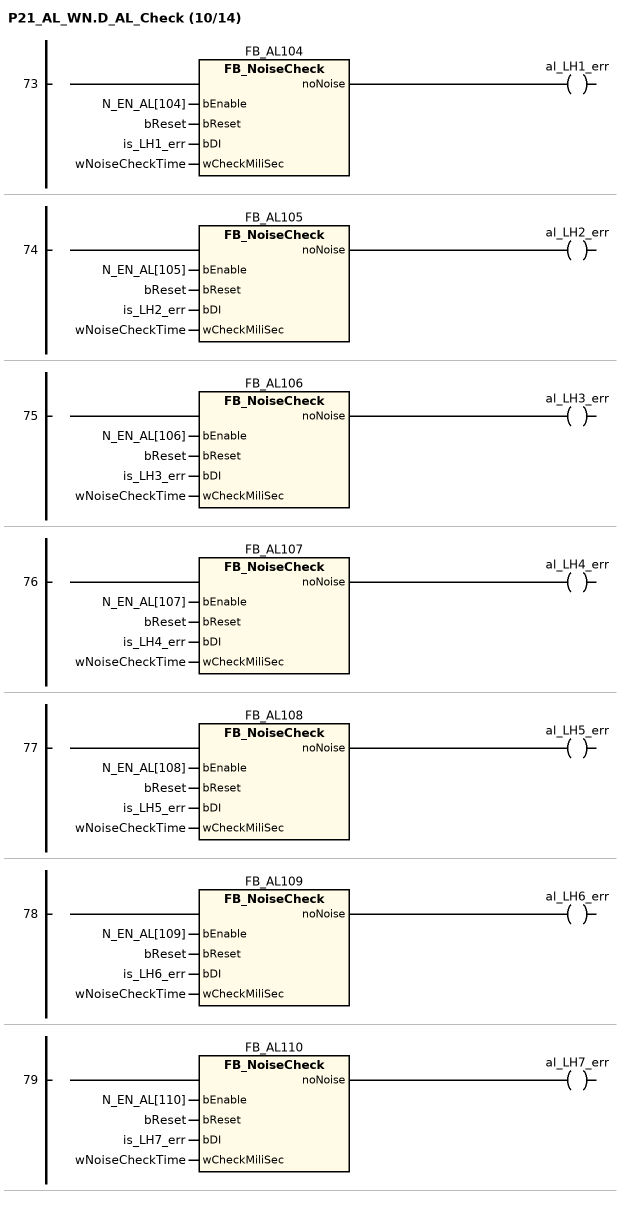
// NETWORK 73
FB_AL104(bEnable := N_EN_AL[104], bReset := bReset, bDI := is_LH1_err, wCheckMiliSec := wNoiseCheckTime); // FB_NoiseCheck
al_LH1_err := FB_AL104.noNoise;

// NETWORK 74
FB_AL105(bEnable := N_EN_AL[105], bReset := bReset, bDI := is_LH2_err, wCheckMiliSec := wNoiseCheckTime); // FB_NoiseCheck
al_LH2_err := FB_AL105.noNoise;

// NETWORK 75
FB_AL106(bEnable := N_EN_AL[106], bReset := bReset, bDI := is_LH3_err, wCheckMiliSec := wNoiseCheckTime); // FB_NoiseCheck
al_LH3_err := FB_AL106.noNoise;

// NETWORK 76
FB_AL107(bEnable := N_EN_AL[107], bReset := bReset, bDI := is_LH4_err, wCheckMiliSec := wNoiseCheckTime); // FB_NoiseCheck
al_LH4_err := FB_AL107.noNoise;

// NETWORK 77
FB_AL108(bEnable := N_EN_AL[108], bReset := bReset, bDI := is_LH5_err, wCheckMiliSec := wNoiseCheckTime); // FB_NoiseCheck
al_LH5_err := FB_AL108.noNoise;

// NETWORK 78
FB_AL109(bEnable := N_EN_AL[109], bReset := bReset, bDI := is_LH6_err, wCheckMiliSec := wNoiseCheckTime); // FB_NoiseCheck
al_LH6_err := FB_AL109.noNoise;

// NETWORK 79
FB_AL110(bEnable := N_EN_AL[110], bReset := bReset, bDI := is_LH7_err, wCheckMiliSec := wNoiseCheckTime); // FB_NoiseCheck
al_LH7_err := FB_AL110.noNoise;

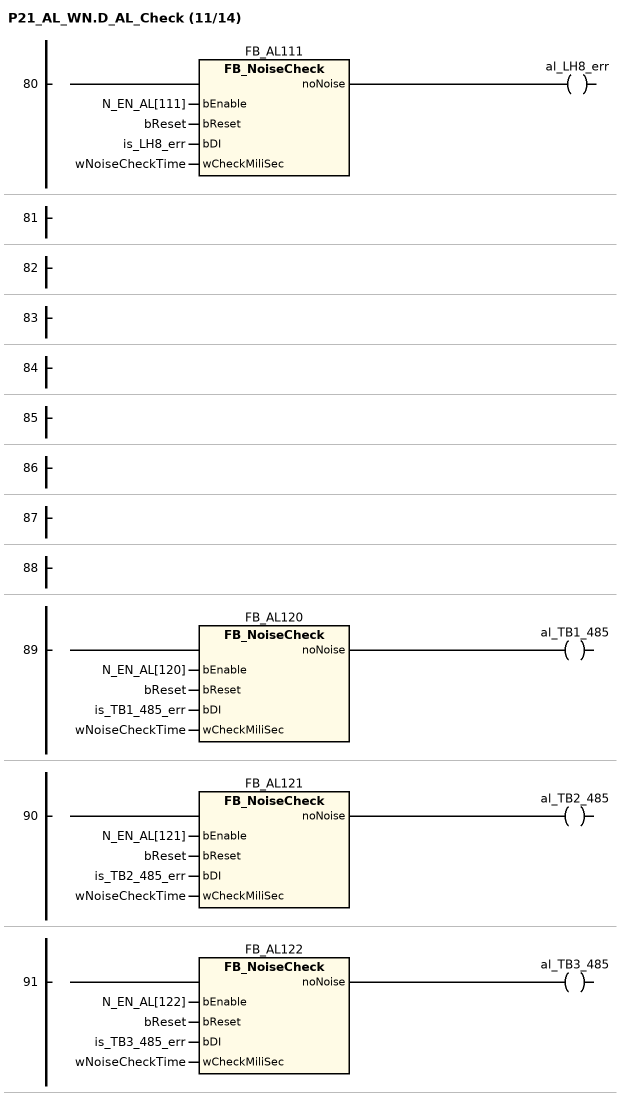
// NETWORK 80
FB_AL111(bEnable := N_EN_AL[111], bReset := bReset, bDI := is_LH8_err, wCheckMiliSec := wNoiseCheckTime); // FB_NoiseCheck
al_LH8_err := FB_AL111.noNoise;

// NETWORK 81

// NETWORK 82

// NETWORK 83

// NETWORK 84

// NETWORK 85

// NETWORK 86

// NETWORK 87

// NETWORK 88

// NETWORK 89
FB_AL120(bEnable := N_EN_AL[120], bReset := bReset, bDI := is_TB1_485_err, wCheckMiliSec := wNoiseCheckTime); // FB_NoiseCheck
al_TB1_485 := FB_AL120.noNoise;

// NETWORK 90
FB_AL121(bEnable := N_EN_AL[121], bReset := bReset, bDI := is_TB2_485_err, wCheckMiliSec := wNoiseCheckTime); // FB_NoiseCheck
al_TB2_485 := FB_AL121.noNoise;

// NETWORK 91
FB_AL122(bEnable := N_EN_AL[122], bReset := bReset, bDI := is_TB3_485_err, wCheckMiliSec := wNoiseCheckTime); // FB_NoiseCheck
al_TB3_485 := FB_AL122.noNoise;

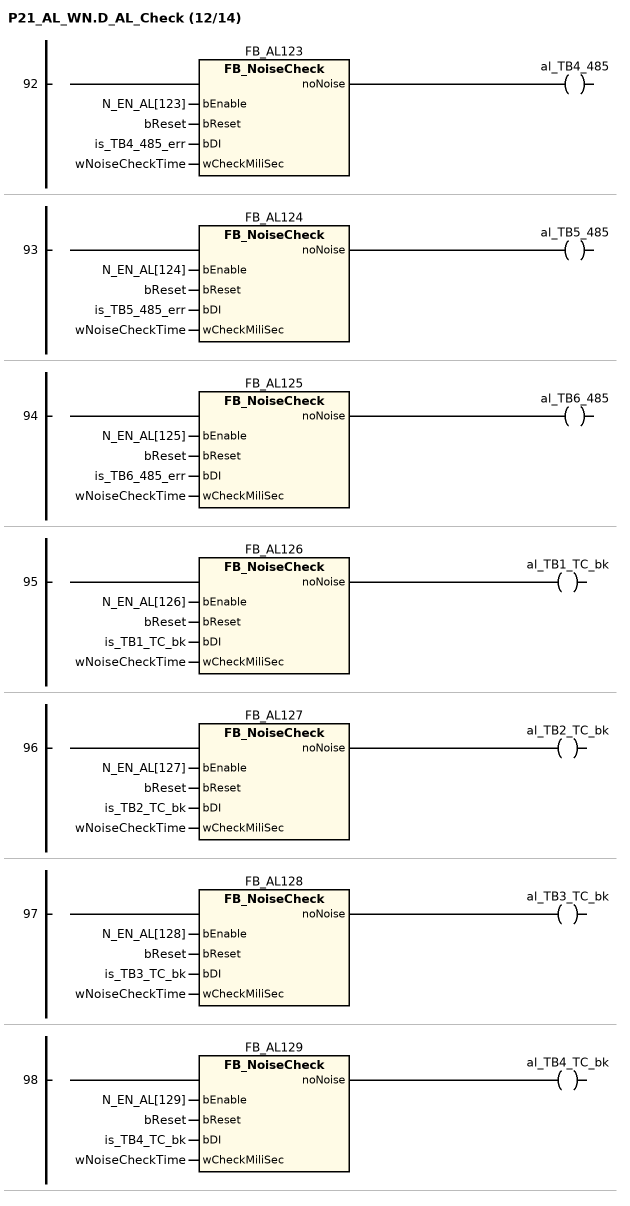
// NETWORK 92
FB_AL123(bEnable := N_EN_AL[123], bReset := bReset, bDI := is_TB4_485_err, wCheckMiliSec := wNoiseCheckTime); // FB_NoiseCheck
al_TB4_485 := FB_AL123.noNoise;

// NETWORK 93
FB_AL124(bEnable := N_EN_AL[124], bReset := bReset, bDI := is_TB5_485_err, wCheckMiliSec := wNoiseCheckTime); // FB_NoiseCheck
al_TB5_485 := FB_AL124.noNoise;

// NETWORK 94
FB_AL125(bEnable := N_EN_AL[125], bReset := bReset, bDI := is_TB6_485_err, wCheckMiliSec := wNoiseCheckTime); // FB_NoiseCheck
al_TB6_485 := FB_AL125.noNoise;

// NETWORK 95
FB_AL126(bEnable := N_EN_AL[126], bReset := bReset, bDI := is_TB1_TC_bk, wCheckMiliSec := wNoiseCheckTime); // FB_NoiseCheck
al_TB1_TC_bk := FB_AL126.noNoise;

// NETWORK 96
FB_AL127(bEnable := N_EN_AL[127], bReset := bReset, bDI := is_TB2_TC_bk, wCheckMiliSec := wNoiseCheckTime); // FB_NoiseCheck
al_TB2_TC_bk := FB_AL127.noNoise;

// NETWORK 97
FB_AL128(bEnable := N_EN_AL[128], bReset := bReset, bDI := is_TB3_TC_bk, wCheckMiliSec := wNoiseCheckTime); // FB_NoiseCheck
al_TB3_TC_bk := FB_AL128.noNoise;

// NETWORK 98
FB_AL129(bEnable := N_EN_AL[129], bReset := bReset, bDI := is_TB4_TC_bk, wCheckMiliSec := wNoiseCheckTime); // FB_NoiseCheck
al_TB4_TC_bk := FB_AL129.noNoise;

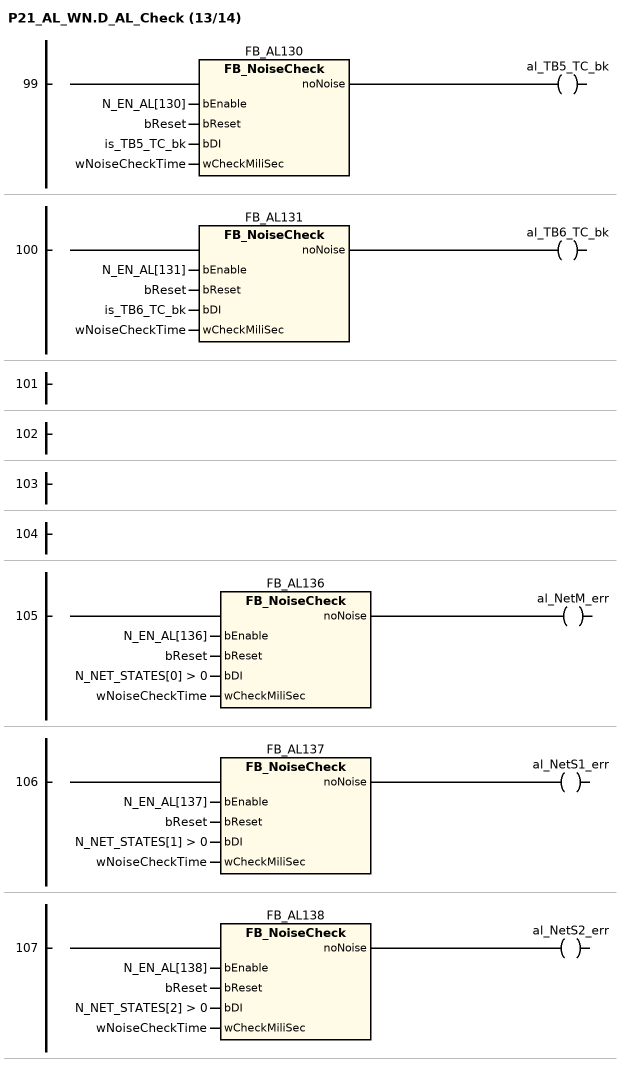
// NETWORK 99
FB_AL130(bEnable := N_EN_AL[130], bReset := bReset, bDI := is_TB5_TC_bk, wCheckMiliSec := wNoiseCheckTime); // FB_NoiseCheck
al_TB5_TC_bk := FB_AL130.noNoise;

// NETWORK 100
FB_AL131(bEnable := N_EN_AL[131], bReset := bReset, bDI := is_TB6_TC_bk, wCheckMiliSec := wNoiseCheckTime); // FB_NoiseCheck
al_TB6_TC_bk := FB_AL131.noNoise;

// NETWORK 101

// NETWORK 102

// NETWORK 103

// NETWORK 104

// NETWORK 105
FB_AL136(
    bEnable := N_EN_AL[136],
    bReset := bReset,
    bDI := N_NET_STATES[0] > 0,
    wCheckMiliSec := wNoiseCheckTime); // FB_NoiseCheck
al_NetM_err := FB_AL136.noNoise;

// NETWORK 106
FB_AL137(
    bEnable := N_EN_AL[137],
    bReset := bReset,
    bDI := N_NET_STATES[1] > 0,
    wCheckMiliSec := wNoiseCheckTime); // FB_NoiseCheck
al_NetS1_err := FB_AL137.noNoise;

// NETWORK 107
FB_AL138(
    bEnable := N_EN_AL[138],
    bReset := bReset,
    bDI := N_NET_STATES[2] > 0,
    wCheckMiliSec := wNoiseCheckTime); // FB_NoiseCheck
al_NetS2_err := FB_AL138.noNoise;

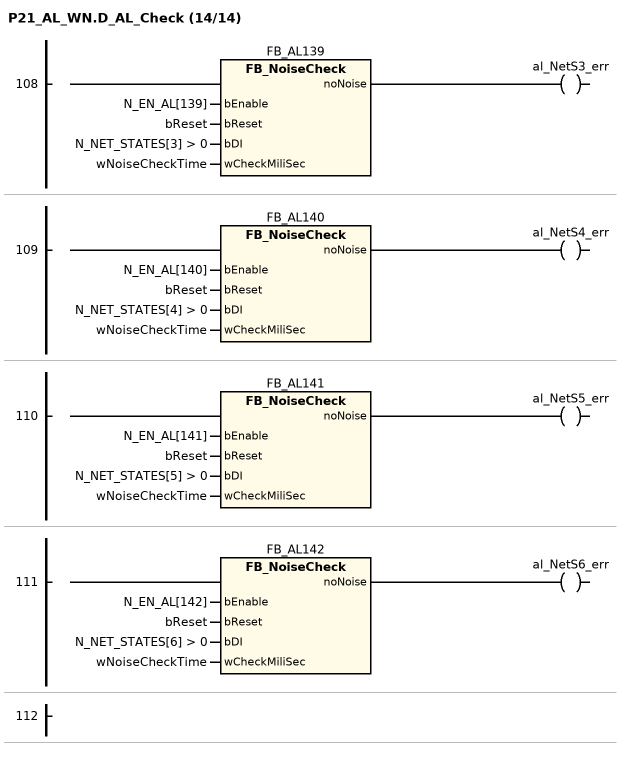
// NETWORK 108
FB_AL139(
    bEnable := N_EN_AL[139],
    bReset := bReset,
    bDI := N_NET_STATES[3] > 0,
    wCheckMiliSec := wNoiseCheckTime); // FB_NoiseCheck
al_NetS3_err := FB_AL139.noNoise;

// NETWORK 109
FB_AL140(
    bEnable := N_EN_AL[140],
    bReset := bReset,
    bDI := N_NET_STATES[4] > 0,
    wCheckMiliSec := wNoiseCheckTime); // FB_NoiseCheck
al_NetS4_err := FB_AL140.noNoise;

// NETWORK 110
FB_AL141(
    bEnable := N_EN_AL[141],
    bReset := bReset,
    bDI := N_NET_STATES[5] > 0,
    wCheckMiliSec := wNoiseCheckTime); // FB_NoiseCheck
al_NetS5_err := FB_AL141.noNoise;

// NETWORK 111
FB_AL142(
    bEnable := N_EN_AL[142],
    bReset := bReset,
    bDI := N_NET_STATES[6] > 0,
    wCheckMiliSec := wNoiseCheckTime); // FB_NoiseCheck
al_NetS6_err := FB_AL142.noNoise;

// NETWORK 112
END_ACTION

ACTION D_WN_Check:
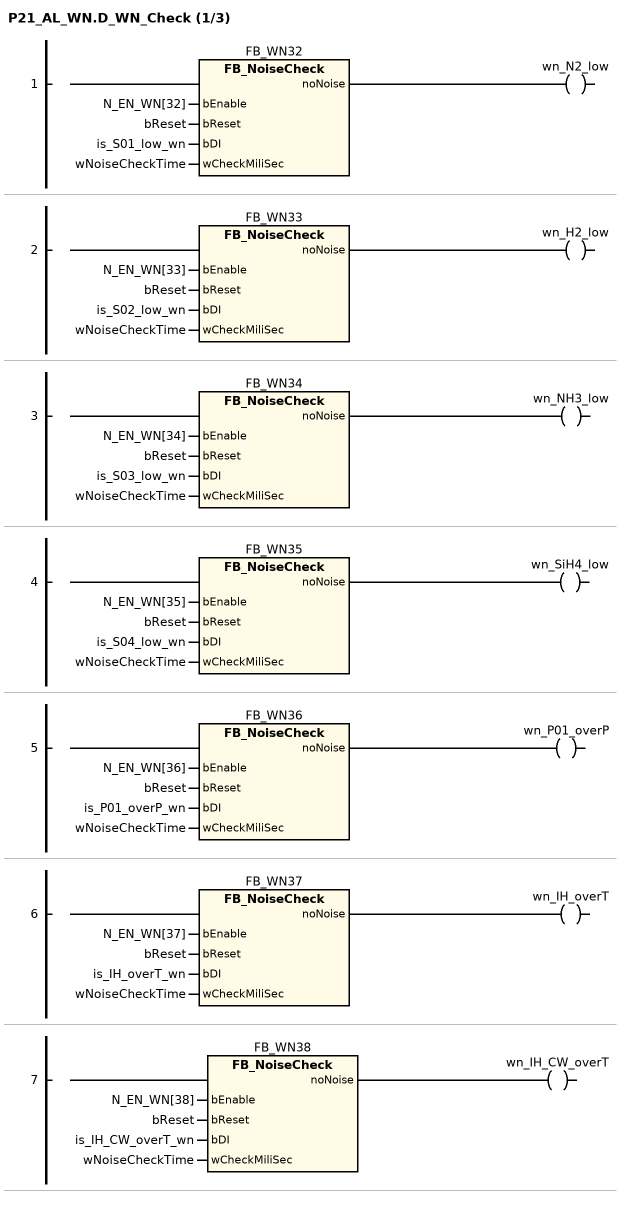
// NETWORK 1
FB_WN32(bEnable := N_EN_WN[32], bReset := bReset, bDI := is_S01_low_wn, wCheckMiliSec := wNoiseCheckTime); // FB_NoiseCheck
wn_N2_low := FB_WN32.noNoise;

// NETWORK 2
FB_WN33(bEnable := N_EN_WN[33], bReset := bReset, bDI := is_S02_low_wn, wCheckMiliSec := wNoiseCheckTime); // FB_NoiseCheck
wn_H2_low := FB_WN33.noNoise;

// NETWORK 3
FB_WN34(bEnable := N_EN_WN[34], bReset := bReset, bDI := is_S03_low_wn, wCheckMiliSec := wNoiseCheckTime); // FB_NoiseCheck
wn_NH3_low := FB_WN34.noNoise;

// NETWORK 4
FB_WN35(bEnable := N_EN_WN[35], bReset := bReset, bDI := is_S04_low_wn, wCheckMiliSec := wNoiseCheckTime); // FB_NoiseCheck
wn_SiH4_low := FB_WN35.noNoise;

// NETWORK 5
FB_WN36(bEnable := N_EN_WN[36], bReset := bReset, bDI := is_P01_overP_wn, wCheckMiliSec := wNoiseCheckTime); // FB_NoiseCheck
wn_P01_overP := FB_WN36.noNoise;

// NETWORK 6
FB_WN37(bEnable := N_EN_WN[37], bReset := bReset, bDI := is_IH_overT_wn, wCheckMiliSec := wNoiseCheckTime); // FB_NoiseCheck
wn_IH_overT := FB_WN37.noNoise;

// NETWORK 7
FB_WN38(bEnable := N_EN_WN[38], bReset := bReset, bDI := is_IH_CW_overT_wn, wCheckMiliSec := wNoiseCheckTime); // FB_NoiseCheck
wn_IH_CW_overT := FB_WN38.noNoise;

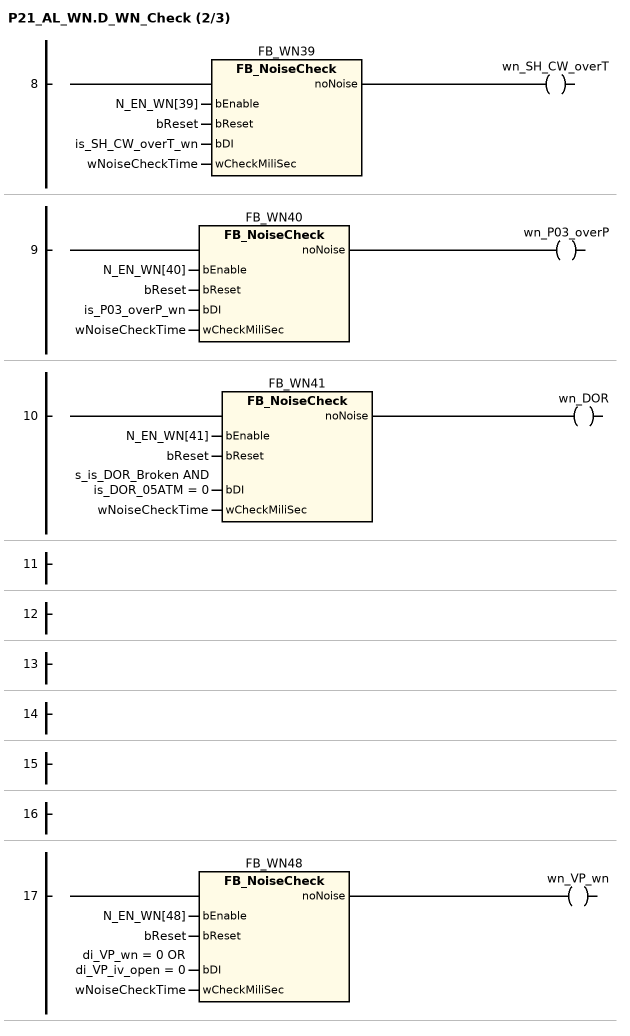
// NETWORK 8
FB_WN39(bEnable := N_EN_WN[39], bReset := bReset, bDI := is_SH_CW_overT_wn, wCheckMiliSec := wNoiseCheckTime); // FB_NoiseCheck
wn_SH_CW_overT := FB_WN39.noNoise;

// NETWORK 9
FB_WN40(bEnable := N_EN_WN[40], bReset := bReset, bDI := is_P03_overP_wn, wCheckMiliSec := wNoiseCheckTime); // FB_NoiseCheck
wn_P03_overP := FB_WN40.noNoise;

// NETWORK 10
FB_WN41(
    bEnable := N_EN_WN[41],
    bReset := bReset,
    bDI := s_is_DOR_Broken AND is_DOR_05ATM = 0,
    wCheckMiliSec := wNoiseCheckTime); // FB_NoiseCheck
wn_DOR := FB_WN41.noNoise;

// NETWORK 11

// NETWORK 12

// NETWORK 13

// NETWORK 14

// NETWORK 15

// NETWORK 16

// NETWORK 17
FB_WN48(
    bEnable := N_EN_WN[48],
    bReset := bReset,
    bDI := di_VP_wn = 0 OR di_VP_iv_open = 0,
    wCheckMiliSec := wNoiseCheckTime); // FB_NoiseCheck
wn_VP_wn := FB_WN48.noNoise;

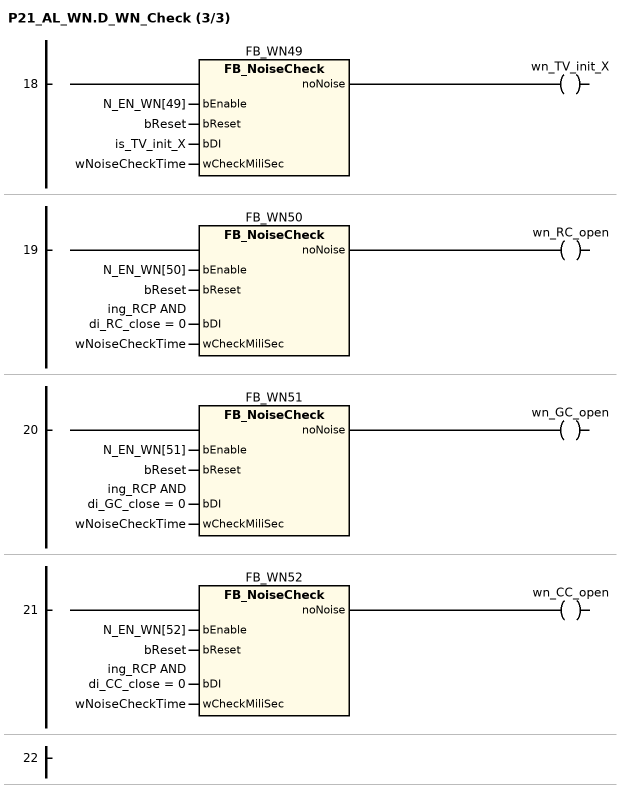
// NETWORK 18
FB_WN49(bEnable := N_EN_WN[49], bReset := bReset, bDI := is_TV_init_X, wCheckMiliSec := wNoiseCheckTime); // FB_NoiseCheck
wn_TV_init_X := FB_WN49.noNoise;

// NETWORK 19
FB_WN50(
    bEnable := N_EN_WN[50],
    bReset := bReset,
    bDI := ing_RCP AND di_RC_close = 0,
    wCheckMiliSec := wNoiseCheckTime); // FB_NoiseCheck
wn_RC_open := FB_WN50.noNoise;

// NETWORK 20
FB_WN51(
    bEnable := N_EN_WN[51],
    bReset := bReset,
    bDI := ing_RCP AND di_GC_close = 0,
    wCheckMiliSec := wNoiseCheckTime); // FB_NoiseCheck
wn_GC_open := FB_WN51.noNoise;

// NETWORK 21
FB_WN52(
    bEnable := N_EN_WN[52],
    bReset := bReset,
    bDI := ing_RCP AND di_CC_close = 0,
    wCheckMiliSec := wNoiseCheckTime); // FB_NoiseCheck
wn_CC_open := FB_WN52.noNoise;

// NETWORK 22
END_ACTION

END_PROGRAM

(* stored: Version 1.1.0.1, ProductVersion 3.1.4024.12
   POU P21_AL_WN: Id {77d66401-4d3a-4af3-b7dc-dd9f22e3f7db}, SpecialFunc None
   Action A_AL_WN_Check: Id {96cac0c5-1bbc-421a-8596-ef8c897b1e0d}
   Action Cause_N_Effect: Id {2442577f-08c4-42c0-9927-0fbaf1993cbb}
   Action D_AL_Check: Id {2bc11194-92ec-4078-a0e5-e363314e3c8d}
   Action D_WN_Check: Id {7d2dbb27-5370-4579-92af-8d4635b4bd19} *)
